(* CODESYS project boiler22.project
   Title: boiler21
   Version: 0.0.0.1

Project tree, tasks and I/O mapping:
  MyController : TM241CE40R, Schneider Electric, order no. TM241CE40R, version 4.0.2.20
    application Application
      libraries: Toolbox, 2.1.0.0 (Schneider Electric); Util, 3.5.1.0 (System); ModbusTCPIOScanner, 1.0.0.4 (Schneider Electric); SysTimeCore, 3.4.1.20 (System)
      task MAST (freewheeling, priority 1, watchdog 100 ms x 1) calls parmStore, service, main, SafeTmr
      task Analog (cyclic, interval t#100ms, priority 2) calls Analog, control
      task calcStat (cyclic, interval t#5s, priority 3) calls calcEnergy
      function HiddenPOU [ST]
      global variables GVL
      Prog/
        program main [ST]
        program Analog [FBD]
        program control [FBD]
        program SafeTmr [FBD]
        function block dualpid [ST]
        function getEnthalpy [ST]
        program service [ST]
        program calcEnergy [ST]
        function getDensity [ST]
        program parmStore [ST]
        function expo [ST]
      RecipeManager
      Symbols
      global variables PersistentVars
    DI : Digital Inputs, Schneider Electric, version 4.0.2.20
        input  xDrumLH2 : BOOL  // IDW0.I0
        input  xDrumLH1 : BOOL  // IDW0.I1
        input  xDrumLl1 : BOOL  // IDW0.I2
        input  xDrumLl2 : BOOL  // IDW0.I3
        input  xGasManOpen : BOOL  // IDW0.I4
        input  xRes1 : BOOL  // IDW0.I5
        input  xRes2 : BOOL  // IDW0.I6
        input  xDrumPh : BOOL  // IDW0.I7
        input  xGasPl : BOOL  // IDW0.I8
        input  xGasPh : BOOL  // IDW0.I9
        input  xAirPl : BOOL  // IDW0.I10
        input  xVacPl : BOOL  // IDW0.I11
        input  xBump : BOOL  // IDW0.I12
        input  xFire1 : BOOL  // IDW0.I13
        input  xTight : BOOL  // IDW0.I14
        input  xSafeOn : BOOL  // IDW0.I15
        input  xStartBn : BOOL  // IDW0.I16
        input  xStopBn : BOOL  // IDW0.I17
        input  xAlarmBn : BOOL  // IDW0.I18
        input  xGasAuto : BOOL  // IDW0.I19
        input  xTermAuto : BOOL  // IDW0.I20
        input  xPumpAuto : BOOL  // IDW0.I21
        input  xExhAuto : BOOL  // IDW0.I22
        input  xFanAuto : BOOL  // IDW0.I23
        unmapped channels: IDW0, IB1
    DQ : Digital Outputs, Schneider Electric, version 4.0.2.20
        output yTermOpen : BOOL  // QW0.Q0
        output yTermClose : BOOL  // QW0.Q1
        output ySuppOpen : BOOL  // QW0.Q2
        output ySuppClose : BOOL  // QW0.Q3
        output yCutofVal : BOOL  // QW0.Q4
        output yBurnerVal : BOOL  // QW0.Q5
        output ySafeVal : BOOL  // QW0.Q6
        output yLitherVal : BOOL  // QW0.Q7
        output yStartFan : BOOL  // QW0.Q8
        output yStartPump : BOOL  // QW0.Q9
        output yGasOpen : BOOL  // QW0.Q10
        output yGasClose : BOOL  // QW0.Q11
        output yPlcStop : BOOL  // QW0.Q12
        output yLamp : BOOL  // QW0.Q13
        output ySerena : BOOL  // QW0.Q14
        output yIgniter : BOOL  // QW0.Q15
        unmapped channels: QW0, QB1
    Counters : Counters, Schneider Electric, version 4.0.2.20
    Pulse_Generators : Pulse Generators, Schneider Electric, version 4.0.2.20
    Cartridge_1 : Cartridge, Schneider Electric, version 4.0.2.20
    Cartridge_2 : Cartridge, Schneider Electric, version 4.0.2.20
    IO_Bus : IO bus - TM3, Schneider Electric, version 4.0.2.20
      Module_2 : TM3AQ4/G, Schneider Electric, order no. TM3AQ4/G, version 1.0.0.10
          settings: KPI Configuration.KPI Configuration[0] = 19; KPI Configuration.KPI Configuration[1] = 19; KPI Configuration.KPI Configuration[2] = 19; KPI Configuration.KPI Configuration[3] = 19; KPI Configuration.KPI Configuration[5] = 0; KPI Configuration.KPI Configuration[7] = 0; KPI Configuration.KPI Configuration[9] = 0; KPI Configuration.KPI Configuration[11] = 0; KPI Configuration.KPI Configuration[12] = 160; KPI Configuration.KPI Configuration[13] = 15; KPI Configuration.KPI Configuration[14] = 160; KPI Configuration.KPI Configuration[15] = 15; KPI Configuration.KPI Configuration[16] = 160; KPI Configuration.KPI Configuration[17] = 15; KPI Configuration.KPI Configuration[18] = 160; KPI Configuration.KPI Configuration[19] = 15
          output Out1 : INT  // QW0
          output Out2 : INT  // QW1
          output Out3 : INT  // QW2
          output Out4 : INT  // QW3
          input  ibModule_2_IBStatusQW0 : BYTE  // IBStatusQW0
          input  ibModule_2_IBStatusQW1 : BYTE  // IBStatusQW1
          input  ibModule_2_IBStatusQW2 : BYTE  // IBStatusQW2
          input  ibModule_2_IBStatusQW3 : BYTE  // IBStatusQW3
      Module_3 : TM3AI8/G, Schneider Electric, order no. TM3AI8/G, version 1.0.0.12
          settings: KPI Configuration.KPI Configuration[0] = 35; KPI Configuration.KPI Configuration[1] = 35; KPI Configuration.KPI Configuration[2] = 35; KPI Configuration.KPI Configuration[3] = 35; KPI Configuration.KPI Configuration[4] = 35; KPI Configuration.KPI Configuration[5] = 35; KPI Configuration.KPI Configuration[6] = 35; KPI Configuration.KPI Configuration[7] = 35; KPI Configuration.KPI Configuration[9] = 0; KPI Configuration.KPI Configuration[11] = 0; KPI Configuration.KPI Configuration[13] = 0; KPI Configuration.KPI Configuration[15] = 0; KPI Configuration.KPI Configuration[17] = 0; KPI Configuration.KPI Configuration[19] = 0; KPI Configuration.KPI Configuration[21] = 0; KPI Configuration.KPI Configuration[23] = 0; KPI Configuration.KPI Configuration[24] = 160; KPI Configuration.KPI Configuration[25] = 15; KPI Configuration.KPI Configuration[26] = 160; KPI Configuration.KPI Configuration[27] = 15; KPI Configuration.KPI Configuration[28] = 160; KPI Configuration.KPI Configuration[29] = 15; KPI Configuration.KPI Configuration[30] = 160; KPI Configuration.KPI Configuration[31] = 15; KPI Configuration.KPI Configuration[32] = 160; KPI Configuration.KPI Configuration[33] = 15; KPI Configuration.KPI Configuration[34] = 160; KPI Configuration.KPI Configuration[35] = 15; KPI Configuration.KPI Configuration[36] = 160; KPI Configuration.KPI Configuration[37] = 15; KPI Configuration.KPI Configuration[38] = 160; KPI Configuration.KPI Configuration[39] = 15
          input  AI000 : INT  // IW0
          input  AI001 : INT  // IW1
          input  AI002 : INT  // IW2
          input  AI003 : INT  // IW3
          input  AI004 : INT  // IW4
          input  AI005 : INT  // IW5
          input  AI006 : INT  // IW6
          input  AI007 : INT  // IW7
          input  ibModule_3_IBStatusIW0 : BYTE  // IBStatusIW0
          input  ibModule_3_IBStatusIW1 : BYTE  // IBStatusIW1
          input  ibModule_3_IBStatusIW2 : BYTE  // IBStatusIW2
          input  ibModule_3_IBStatusIW3 : BYTE  // IBStatusIW3
          input  ibModule_3_IBStatusIW4 : BYTE  // IBStatusIW4
          input  ibModule_3_IBStatusIW5 : BYTE  // IBStatusIW5
          input  ibModule_3_IBStatusIW6 : BYTE  // IBStatusIW6
          input  ibModule_3_IBStatusIW7 : BYTE  // IBStatusIW7
      Module_4 : TM3AI8/G, Schneider Electric, order no. TM3AI8/G, version 1.0.0.12
          settings: KPI Configuration.KPI Configuration[0] = 35; KPI Configuration.KPI Configuration[1] = 35; KPI Configuration.KPI Configuration[2] = 35; KPI Configuration.KPI Configuration[3] = 35; KPI Configuration.KPI Configuration[4] = 35; KPI Configuration.KPI Configuration[5] = 35; KPI Configuration.KPI Configuration[6] = 35; KPI Configuration.KPI Configuration[7] = 35; KPI Configuration.KPI Configuration[9] = 0; KPI Configuration.KPI Configuration[11] = 0; KPI Configuration.KPI Configuration[13] = 0; KPI Configuration.KPI Configuration[15] = 0; KPI Configuration.KPI Configuration[17] = 0; KPI Configuration.KPI Configuration[19] = 0; KPI Configuration.KPI Configuration[21] = 0; KPI Configuration.KPI Configuration[23] = 0; KPI Configuration.KPI Configuration[24] = 160; KPI Configuration.KPI Configuration[25] = 15; KPI Configuration.KPI Configuration[26] = 160; KPI Configuration.KPI Configuration[27] = 15; KPI Configuration.KPI Configuration[28] = 160; KPI Configuration.KPI Configuration[29] = 15; KPI Configuration.KPI Configuration[30] = 160; KPI Configuration.KPI Configuration[31] = 15; KPI Configuration.KPI Configuration[32] = 160; KPI Configuration.KPI Configuration[33] = 15; KPI Configuration.KPI Configuration[34] = 160; KPI Configuration.KPI Configuration[35] = 15; KPI Configuration.KPI Configuration[36] = 160; KPI Configuration.KPI Configuration[37] = 15; KPI Configuration.KPI Configuration[38] = 160; KPI Configuration.KPI Configuration[39] = 15
          input  AI010 : INT  // IW0
          input  AI011 : INT  // IW1
          input  AI012 : INT  // IW2
          input  AI013 : INT  // IW3
          input  AI014 : INT  // IW4
          input  AI015 : INT  // IW5
          input  AI016 : INT  // IW6
          input  AI017 : INT  // IW7
          input  ibModule_4_IBStatusIW0 : BYTE  // IBStatusIW0
          input  ibModule_4_IBStatusIW1 : BYTE  // IBStatusIW1
          input  ibModule_4_IBStatusIW2 : BYTE  // IBStatusIW2
          input  ibModule_4_IBStatusIW3 : BYTE  // IBStatusIW3
          input  ibModule_4_IBStatusIW4 : BYTE  // IBStatusIW4
          input  ibModule_4_IBStatusIW5 : BYTE  // IBStatusIW5
          input  ibModule_4_IBStatusIW6 : BYTE  // IBStatusIW6
          input  ibModule_4_IBStatusIW7 : BYTE  // IBStatusIW7
      Module_5 : TM3AI8/G, Schneider Electric, order no. TM3AI8/G, version 1.0.0.12
          settings: KPI Configuration.KPI Configuration[0] = 35; KPI Configuration.KPI Configuration[1] = 35; KPI Configuration.KPI Configuration[2] = 35; KPI Configuration.KPI Configuration[3] = 35; KPI Configuration.KPI Configuration[4] = 35; KPI Configuration.KPI Configuration[5] = 35; KPI Configuration.KPI Configuration[6] = 35; KPI Configuration.KPI Configuration[7] = 35; KPI Configuration.KPI Configuration[9] = 0; KPI Configuration.KPI Configuration[11] = 0; KPI Configuration.KPI Configuration[13] = 0; KPI Configuration.KPI Configuration[15] = 0; KPI Configuration.KPI Configuration[17] = 0; KPI Configuration.KPI Configuration[19] = 0; KPI Configuration.KPI Configuration[21] = 0; KPI Configuration.KPI Configuration[23] = 0; KPI Configuration.KPI Configuration[24] = 160; KPI Configuration.KPI Configuration[25] = 15; KPI Configuration.KPI Configuration[26] = 160; KPI Configuration.KPI Configuration[27] = 15; KPI Configuration.KPI Configuration[28] = 160; KPI Configuration.KPI Configuration[29] = 15; KPI Configuration.KPI Configuration[30] = 160; KPI Configuration.KPI Configuration[31] = 15; KPI Configuration.KPI Configuration[32] = 160; KPI Configuration.KPI Configuration[33] = 15; KPI Configuration.KPI Configuration[34] = 160; KPI Configuration.KPI Configuration[35] = 15; KPI Configuration.KPI Configuration[36] = 160; KPI Configuration.KPI Configuration[37] = 15; KPI Configuration.KPI Configuration[38] = 160; KPI Configuration.KPI Configuration[39] = 15
          input  AI020 : INT  // IW0
          input  AI021 : INT  // IW1
          input  AI022 : INT  // IW2
          input  AI023 : INT  // IW3
          input  AI024 : INT  // IW4
          input  AI025 : INT  // IW5
          input  AI026 : INT  // IW6
          input  AI027 : INT  // IW7
          input  ibModule_5_IBStatusIW0 : BYTE  // IBStatusIW0
          input  ibModule_5_IBStatusIW1 : BYTE  // IBStatusIW1
          input  ibModule_5_IBStatusIW2 : BYTE  // IBStatusIW2
          input  ibModule_5_IBStatusIW3 : BYTE  // IBStatusIW3
          input  ibModule_5_IBStatusIW4 : BYTE  // IBStatusIW4
          input  ibModule_5_IBStatusIW5 : BYTE  // IBStatusIW5
          input  ibModule_5_IBStatusIW6 : BYTE  // IBStatusIW6
          input  ibModule_5_IBStatusIW7 : BYTE  // IBStatusIW7
    COM_Bus : COM bus, Schneider Electric, version 4.0.2.20
    Ethernet_1 : Ethernet Network, Schneider Electric, version 4.0.2.20
        settings: IPAddress = [192, 168, 15, 152]; SubnetMask = [255, 255, 255, 0]; GatewayAddress = [192, 168, 15, 1]; DeviceName = 'boiler2'; WebServer = FALSE; FTP Server = FALSE; SoMachine Protocol = TRUE; Modbus Server = TRUE; NetManage Protocol = FALSE; SNMP protocol = FALSE; Enable Routing = FALSE; WebVisu protocol = FALSE
    Serial_Line_1 : Serial line, Schneider Electric, version 4.0.2.20
      Modbus_Manager : Modbus Manager, Schneider Electric, version 4.0.0.2
    Serial_Line_2 : Serial line, Schneider Electric, version 4.0.2.20
      Modbus_IOScanner : Modbus IOScanner, Schneider Electric, version 3.5.3.6
        drvFan : Generic Modbus Slave, Schneider Electric, version 3.5.3.6
            settings: SlaveAddress = 12; ResponseTimeout = 1000; Channel 1.Function Code = 3; Channel 1.Read Offset = 16#0008; Channel 1.Read Length = 1; Channel 1.Write Offset = 0; Channel 1.Write Length = 0; Channel 1.Cycle Time = 0; Channel 2.Function Code = 3; Channel 2.Read Offset = 16#00C8; Channel 2.Read Length = 8; Channel 2.Write Offset = 0; Channel 2.Write Length = 0; Channel 2.Cycle Time = 0
            input  fanStatus : WORD  // Channel 1.Channel 1[0]
            input  fan0 : WORD  // Channel 2.Channel 2[0]
            input  fan1 : WORD  // Channel 2.Channel 2[1]
            input  fan2 : WORD  // Channel 2.Channel 2[2]
            input  fan3 : WORD  // Channel 2.Channel 2[3]
            input  fan4 : WORD  // Channel 2.Channel 2[4]
            input  fan5 : WORD  // Channel 2.Channel 2[5]
            input  fan6 : WORD  // Channel 2.Channel 2[6]
            input  fan7 : WORD  // Channel 2.Channel 2[7]
            unmapped channels: Channel 1, Channel 2
        PD150 : Generic Modbus Slave, Schneider Electric, version 3.5.3.6
            settings: SlaveAddress = 16; ResponseTimeout = 1000; Channel 1.Function Code = 3; Channel 1.Read Offset = 16#0013; Channel 1.Read Length = 2; Channel 1.Write Offset = 0; Channel 1.Write Length = 0; Channel 1.Cycle Time = 0
            input  pdi1 : WORD  // Channel 1.Channel 1[0]
            input  pdi2 : WORD  // Channel 1.Channel 1[1]
            unmapped channels: Channel 1
        drvPump : Generic Modbus Slave, Schneider Electric, version 3.5.3.6
            settings: SlaveAddress = 10; ResponseTimeout = 1000; Channel 1.Function Code = 3; Channel 1.Read Offset = 16#0066; Channel 1.Read Length = 8; Channel 1.Write Offset = 0; Channel 1.Write Length = 0; Channel 1.Cycle Time = 0; Channel 2.Function Code = 2; Channel 2.Read Offset = 16#0000; Channel 2.Read Length = 16; Channel 2.Write Offset = 0; Channel 2.Write Length = 0; Channel 2.Cycle Time = 0
            input  pump0 : WORD  // Channel 1.Channel 1[0]
            input  pump1 : WORD  // Channel 1.Channel 1[1]
            input  pump2 : WORD  // Channel 1.Channel 1[2]
            input  pump3 : WORD  // Channel 1.Channel 1[3]
            input  pump4 : WORD  // Channel 1.Channel 1[4]
            input  pump5 : WORD  // Channel 1.Channel 1[5]
            input  pump6 : WORD  // Channel 1.Channel 1[6]
            input  pump7 : WORD  // Channel 1.Channel 1[7]
            input  pumpRun : BOOL  // Channel 2.Channel 2[0].Bit2
            unmapped channels: Channel 1, Channel 2
        drvExh : Generic Modbus Slave, Schneider Electric, version 3.5.3.6
            settings: SlaveAddress = 11; ResponseTimeout = 1000; Channel 1.Function Code = 3; Channel 1.Read Offset = 16#1101; Channel 1.Read Length = 11; Channel 1.Write Offset = 0; Channel 1.Write Length = 0; Channel 1.Cycle Time = 0; Channel 2.Function Code = 3; Channel 2.Read Offset = 16#2100; Channel 2.Read Length = 3; Channel 2.Write Offset = 0; Channel 2.Write Length = 0; Channel 2.Cycle Time = 0
            input  exh0 : WORD  // Channel 1.Channel 1[0]
            input  exh1 : WORD  // Channel 1.Channel 1[1]
            input  exh2 : WORD  // Channel 1.Channel 1[2]
            input  exh3 : WORD  // Channel 1.Channel 1[3]
            input  exh4 : WORD  // Channel 1.Channel 1[4]
            input  exh5 : WORD  // Channel 1.Channel 1[5]
            input  exh6 : WORD  // Channel 1.Channel 1[6]
            input  exh7 : WORD  // Channel 1.Channel 1[7]
            input  exh8 : WORD  // Channel 1.Channel 1[8]
            input  exh9 : WORD  // Channel 1.Channel 1[9]
            input  exh10 : WORD  // Channel 1.Channel 1[10]
            input  exhStatus : WORD  // Channel 2.Channel 2[0]
            unmapped channels: Channel 1, Channel 2
  FdtConnections : FDT Connections, Schneider Electric, version 1.0.0.2
    Modbus_Serial_Line_Manager : Modbus Serial Line Manager, Schneider Electric, version 2.2.5
*)

// MyController/Application/GVL

VAR_GLOBAL
allAM AT %MW0: INT;

AM001 AT %MX0.0: BOOL;
AM002 AT %MX0.1: BOOL;
AM003 AT %MX0.2: BOOL;
AM004 AT %MX0.3: BOOL;
AM005 AT %MX0.4: BOOL;
AM006 AT %MX0.5: BOOL;
AM007 AT %MX0.6: BOOL;
AM008 AT %MX0.7: BOOL;

amGas AT %MX2.0: BOOL := true;
amTerm AT %MX2.1: BOOL := true;
amSupp AT %MX2.2: BOOL := true;

Alm0001 AT %MX4.0: BOOL;
Alm0002 AT %MX4.1: BOOL;
Alm0003 AT %MX4.2: BOOL;
Alm0004 AT %MX4.3: BOOL;
Alm0005 AT %MX4.4: BOOL;
Alm0006 AT %MX4.5: BOOL;
Alm0007 AT %MX4.6: BOOL;
Alm0008 AT %MX4.7: BOOL;
Alm0009 AT %MX5.0: BOOL;
Alm0010 AT %MX5.1: BOOL;
Alm0011 AT %MX5.2: BOOL;
Alm0012 AT %MX5.3: BOOL;
alFire1 AT %MX5.4: BOOL;
alFan AT %MX5.5: BOOL;
alExh AT %MX5.6: BOOL;
alPump AT %MX5.7: BOOL;


alSupport AT %MX6.0: BOOL;
linkPump AT %MX6.1: BOOL;
linkFan AT %MX6.2: BOOL;
linkExh AT %MX6.3: BOOL;
linkPD150 AT %MX6.4: BOOL;
stab1 AT %MX6.5: BOOL;
stab2 AT %MX6.6: BOOL;
stab3 AT %MX6.7: BOOL;
stab4 AT %MX7.0: BOOL;
stab5 AT %MX7.1: BOOL;
xFanRun AT %MX7.2: BOOL;
xExhRun AT %MX7.3: BOOL;
xPumpRun AT %MX7.4: BOOL;
stWait AT %MX7.5: BOOL;
Alert AT %MX7.6: BOOL;
Halt AT %MX7.7: BOOL;

// це треба буде писати зверху
Run AT %MX8.0: BOOL;
Cvit AT %MX10.0: BOOL;
prLock AT %MX12.0: BOOL;
serenaLock AT %MX12.1: BOOL;

bnAll AT %MW7: INT;
bnStart AT %MX14.0: BOOL;
bnStop AT %MX14.1: BOOL;
// список прогодження кроків програми запуску
check0 AT %MX16.0: BOOL;
check1 AT %MX16.1: BOOL;
check2 AT %MX16.2: BOOL;
check3 AT %MX16.3: BOOL;
check4 AT %MX16.4: BOOL;
check5 AT %MX16.5: BOOL;
check6 AT %MX16.6: BOOL;
check7 AT %MX16.7: BOOL;
check8 AT %MX17.0: BOOL;
check9 AT %MX17.1: BOOL;
check10 AT %MX17.2: BOOL;
check11 AT %MX17.3: BOOL;
check12 AT %MX17.4: BOOL;
check13 AT %MX17.5: BOOL;
check14 AT %MX17.6: BOOL;
check15 AT %MX17.7: BOOL;

checkList AT %MW8: UINT;


Pack_lo AT %MW998: WORD;
Pack_hi AT %MW999: WORD;
Pack_v AT %MD499: REAL;

Fgas AT %MD5: REAL;
Fpara AT %MD6: REAL;
Fwater AT %MD7: REAL;
Fair AT %MD8: REAL;
Ldrum AT %MD9: REAL;
Pg15a AT %MD10: REAL;
Ppara AT %MD11: REAL;
Pp7a AT %MD12: REAL;
Tpar AT %MD13: REAL;
Tv3a AT %MD14: REAL;
Tv4a AT %MD15: REAL;
Tk AT %MD16: REAL;
Ta5a AT %MD17: REAL;
Ta6a AT %MD18: REAL;
Tp17a AT %MD19: REAL;
Tp18a AT %MD20: REAL;
Pair AT %MD21: REAL;
Pvac AT %MD22: REAL;
Pv12a AT %MD23: REAL;
gGas AT %MD24: REAL;
gTerm AT %MD25: REAL;
gSupp AT %MD26: REAL;
QO2fume AT %MD27: REAL;
Vx AT %MD28: REAL;

W01 AT %MW10: WORD;
W02 AT %MW11: WORD;

END_VAR

VAR_GLOBAL RETAIN
cPump AT %MD29: REAL;
cFan AT %MD30: REAL;
cExh AT %MD31: REAL;
cGas AT %MD32: REAL;
cTerm AT %MD33: REAL;
cSupport AT %MD34: REAL;
cX AT %MD35: REAL;
END_VAR

VAR_GLOBAL
FanSpeed AT %MD36: REAL;
FanCurrent AT %MD37: REAL;
FanVoltage AT %MD38: REAL;
FanDC AT %MD39: REAL;
PumpSpeed AT %MD40: REAL;
PumpCurrent AT %MD41: REAL;
PumpVoltage AT %MD42: REAL;
PumpDC AT %MD43: REAL;
ExhSpeed AT %MD44: REAL;
ExhCurrent AT %MD45: REAL;
ExhVoltage AT %MD46: REAL;
ExhDC AT %MD47: REAL;

END_VAR

VAR_GLOBAL RETAIN
Sp0001 AT %MD48: REAL;
Sp0002 AT %MD49: REAL;
Sp0003 AT %MD50: REAL;
Sp0004 AT %MD51: REAL;
Sp0005 AT %MD52: REAL;
Sp0006 AT %MD53: REAL;
Sp0007 AT %MD54: REAL;
Sp0008 AT %MD55: REAL;
Sp0009 AT %MD56: REAL;
Sp0010 AT %MW114: UINT;
END_VAR

VAR_GLOBAL


// Кінцевий автомат управління котлом
State AT %MW115: UINT;
stateTight AT %MW116: UINT;
flame AT %MW117: UINT;

pvTVentPre AT %MD400: DWORD;
pvTBlowing AT %MD401: DWORD;
pvFiring AT %MD402: DWORD;
pvStartfeed AT %MD403: DWORD;
pvStartExh AT %MD404: DWORD;
pvStartfan AT %MD405: DWORD;
pvIgniting AT %MD406: DWORD;
pvTVentPost AT %MD407: DWORD;

END_VAR

VAR_GLOBAL RETAIN
backup AT %MW118: UINT;

uptime AT %MD425: REAL;
allPara AT %MD426: REAL;
allGas AT %MD427: REAL;
allWarm AT %MD428: REAL;
allEce AT %MD429: REAL;
hourPara AT %MD430: REAL;
hourGas AT %MD431: REAL;
hourWarm AT %MD432: REAL;
hourEce AT %MD433: REAL;

 
fA000 AT %MW177: UINT;
fA001 AT %MW178: UINT;
fA002 AT %MW179: UINT;
fA003 AT %MW180: UINT;
fA004 AT %MW181: UINT;
fA005 AT %MW182: UINT;
fA006 AT %MW183: UINT;
fA007 AT %MW184: UINT;
fA010 AT %MW185: UINT;
fA011 AT %MW186: UINT;
fA012 AT %MW187: UINT;
fA013 AT %MW188: UINT;
fA014 AT %MW189: UINT;
fA015 AT %MW190: UINT;
fA016 AT %MW191: UINT;
fA017 AT %MW192: UINT;
fA020 AT %MW193: UINT;
fA021 AT %MW194: UINT;
fA022 AT %MW195: UINT;
fA023 AT %MW196: UINT;
fA024 AT %MW197: UINT;
fA025 AT %MW198: UINT;
fA026 AT %MW199: UINT;
fA027 AT %MW200: UINT;

modeGas AT %MW201: UINT;

Kp0001 AT %MD101: REAL;
Ti0001 AT %MD102: REAL;
Td0001 AT %MD103: REAL;
Xmin0001 AT %MD104: REAL;
Xmax0001 AT %MD105: REAL;
Kp0002 AT %MD106: REAL;
Ti0002 AT %MD107: REAL;
Td0002 AT %MD108: REAL;
Xmin0002 AT %MD109: REAL;
Xmax0002 AT %MD110: REAL;
Kp0003 AT %MD111: REAL;
Ti0003 AT %MD112: REAL;
Td0003 AT %MD113: REAL;
Xmin0003 AT %MD114: REAL;
Xmax0003 AT %MD115: REAL;
Kp0004 AT %MD116: REAL;
Ti0004 AT %MD117: REAL;
Td0004 AT %MD118: REAL;
Xmin0004 AT %MD119: REAL;
Xmax0004 AT %MD120: REAL;
Kp0005 AT %MD121: REAL;
Ti0005 AT %MD122: REAL;
Td0005 AT %MD123: REAL;
Xmin0005 AT %MD124: REAL;
Xmax0005 AT %MD125: REAL;
Kp0006 AT %MD126: REAL;
Ti0006 AT %MD127: REAL;
Td0006 AT %MD128: REAL;
Xmin0006 AT %MD129: REAL;
Xmax0006 AT %MD130: REAL;
Kp0007 AT %MD131: REAL;
Ti0007 AT %MD132: REAL;
Td0007 AT %MD133: REAL;
Xmin0007 AT %MD134: REAL;
Xmax0007 AT %MD135: REAL;
Kp0008 AT %MD136: REAL;
Ti0008 AT %MD137: REAL;
Td0008 AT %MD138: REAL;
Xmin0008 AT %MD139: REAL;
Xmax0008 AT %MD140: REAL;
startSP0002 AT %MD141: REAL;

tMeoTerm AT %MD142: REAL;
tMeoGas AT %MD143: REAL;
dGas AT %MD144: REAL;
dTerm AT %MD145: REAL;
dSupport AT %MD146: REAL;
maxS1 AT %MD147: REAL;
maxS2 AT %MD148: REAL;
maxS3 AT %MD149: REAL;
maxS4 AT %MD150: REAL;
maxS5 AT %MD151: REAL;
K2001 AT %MD152: REAL;
startPump AT %MD153: REAL;
startFan AT %MD154: REAL;
startExh AT %MD155: REAL;
startGas AT %MD156: REAL;
startTerm AT %MD157: REAL;
gOffset AT %MD158: REAL;
gGain AT %MD159: REAL;
heatingGas AT %MD160: REAL;
sca_Ppara AT %MD161: REAL;
max_Ppara AT %MD162: REAL;
sca_Tpar AT %MD163: REAL;
max_Tpar AT %MD164: REAL;
sca_Tv3a AT %MD165: REAL;
max_Tv3a AT %MD166: REAL;
sca_Fgas AT %MD167: REAL;
max_Fgas AT %MD168: REAL;
sca_Fpara AT %MD169: REAL;
max_Fpara AT %MD170: REAL;
qgas AT %MD171: REAL;
sca_Fwater AT %MD172: REAL;
max_Fwater AT %MD173: REAL;
gTermOffset AT %MD174: REAL;
gTermGain AT %MD175: REAL;
gSuppOffset AT %MD176: REAL;
gSuppGain AT %MD177: REAL;
Ke0001 AT %MD178: REAL;
Ke0002 AT %MD179: REAL;
Ke0003 AT %MD180: REAL;
Ke0004 AT %MD181: REAL;
Ke0005 AT %MD182: REAL;
Kmix001 AT %MD183: REAL;
Kmix002 AT %MD184: REAL;
Kmix003 AT %MD185: REAL;
Kmix004 AT %MD186: REAL;
Kmix005 AT %MD187: REAL;
Omix001 AT %MD188: REAL;
Omix002 AT %MD189: REAL;
Omix003 AT %MD190: REAL;
Omix004 AT %MD191: REAL;
Omix005 AT %MD192: REAL;
ignSP0002 AT %MD193: REAL;

Tpr0001 AT %MD256: DWORD;
Tpr0002 AT %MD257: DWORD;
Tpr0003 AT %MD258: DWORD;
Tpr0004 AT %MD259: DWORD;
Tpr0005 AT %MD260: DWORD;
Tpr0006 AT %MD261: DWORD;
Tpr0007 AT %MD262: DWORD;
Tpr0008 AT %MD263: DWORD;
Tpr0009 AT %MD264: DWORD;
Tpr0010 AT %MD265: DWORD;
Tpr0011 AT %MD266: DWORD;
Tpr0012 AT %MD267: DWORD;
spTstart AT %MD268: DWORD;
spTVentPre AT %MD269: DWORD;
spTVentPost AT %MD270: DWORD;
spTBlowing AT %MD271: DWORD;
spStartfeed AT %MD272: DWORD;
spStartExh AT %MD273: DWORD;
spStartfan AT %MD274: DWORD;
spIgniting AT %MD275: DWORD;



END_VAR

VAR_GLOBAL
firstStep: BOOL:=TRUE;
	
Xt0001: REAL;
Xt0002: REAL;
Xt0003: REAL;
Xt0004: REAL;
Xt0005: REAL;
Xt0006: REAL;
Xt0007: REAL;
Xt0008: REAL;

tMeo1: TIME;
tMeo2: TIME;
tMeo3: TIME;

enthalpy: REAL;

regO2en: BOOL;
pwmParam: stPwmPara;

p4GasOpen: BOOL;
p4GasClose: BOOL;

END_VAR

VAR_GLOBAL CONSTANT
// таблиця ентальпії пари від 200 до 500 *С з кроком 10*С і від 1000 до 3000 кПа з кроком 500кПа	
enthalpyTab: ARRAY[0..30] OF ARRAY[0..4] OF REAL := [
[2827.5,2795.3,852.6,852.8,853.0],
[2851.5,2822.9,897.8,898.1,898.1],
[2874.9,2849.2,2820.4,943.7,943.9],
[2897.9,2874.7,2849.0,2820.4,990.3],
[2920.5,2899.3,2876.3,2851.0,2823.0],
[2942.8,2923.4,2902.5,2879.9,2855.2],
[2964.8,2947.0,2927.9,2907.5,2885.5],
[2986.7,2970.2,2952.7,2934.1,2914.2],
[3008.3,2993.0,2976.9,2959.8,2941.8],
[3029.9,3015.6,3000.6,2984.9,2968.4],
[3051.3,3037.9,3024.0,3009.4,2994.2],
[3072.7,3060.1,3047.0,3033.4,3019.3],
[3094.0,3082.1,3069.8,3057.1,3044.0],
[3115.3,3104.0,3092.4,3080.5,3068.2],
[3136.5,3125.8,3114.9,3103.6,3092.1],
[3157.7,3147.6,3137.2,3126.6,3115.7],
[3178.9,3169.3,3159.5,3149.6,3139.3],
[3200.2,3191.1,3181.8,3172.4,3162.7],
[3221.5,3212.8,3204.0,3195.0,3185.8],
[3242.8,3234.5,3226.1,3217.5,3208.8],
[3264.0,3256.1,3248.1,3239.9,3231.6],
[3285.3,3277.7,3270.0,3262.2,3254.3],
[3306.6,3299.3,3291.9,3284.5,3276.9],
[3327.9,3320.9,3313.8,3306.7,3299.4],
[3349.3,3342.6,3335.7,3328.9,3321.9],
[3370.7,3364.2,3357.7,3351.0,3344.4],
[3392.1,3385.9,3379.6,3373.2,3366.8],
[3413.8,3407.6,3401.5,3395.4,3389.2],
[3435.1,3429.3,3423.5,3417.5,3411.6],
[3456.7,3451.1,3445.4,3439.7,3434.0],
[3478.3,3472.9,3467.4,3461.9,3456.4]
];	
// питомий обёєм 
spvolTab: ARRAY[0..30] OF ARRAY[0..4] OF REAL := [
[	0.2059	,	0.1324	,	0.001156	,	0.0011555	,	0.001155	],
[	0.2115	,	0.1366	,	0.0011725	,	0.0011719	,	0.0011714	],
[	0.2169	,	0.14	,	0.10211	,	0.0011897	,	0.0011891	],
[	0.2223	,	0.1445	,	0.1053	,	0.08164	,	0.0012084	],
[	0.2275	,	0.1483	,	0.1084	,	0.08439	,	0.06818	],
[	0.2327	,	0.152	,	0.1115	,	0.08701	,	0.07058	],
[	0.2378	,	0.1556	,	0.1144	,	0.08953	,	0.07286	],
[	0.2429	,	0.1592	,	0.1172	,	0.09197	,	0.07504	],
[	0.248	,	0.1627	,	0.12	,	0.09434	,	0.07714	],
[	0.253	,	0.1662	,	0.1228	,	0.09665	,	0.07918	],
[	0.258	,	0.1697	,	0.1255	,	0.09892	,	0.08116	],
[	0.2629	,	0.1731	,	0.1282	,	0.10114	,	0.0831	],
[	0.2678	,	0.1765	,	0.1308	,	0.10334	,	0.085	],
[	0.2727	,	0.1799	,	0.1334	,	0.1055	,	0.08687	],
[	0.2776	,	0.1832	,	0.136	,	0.1076	,	0.08871	],
[	0.2825	,	0.1866	,	0.1386	,	0.1098	,	0.09053	],
[	0.2873	,	0.1899	,	0.1411	,	0.1119	,	0.09232	],
[	0.2921	,	0.1932	,	0.1436	,	0.1139	,	0.0941	],
[	0.297	,	0.1964	,	0.1462	,	0.116	,	0.09586	],
[	0.3018	,	0.1997	,	0.1487	,	0.118	,	0.0976	],
[	0.3066	,	0.203	,	0.1512	,	0.1201	,	0.09933	],
[	0.3113	,	0.2062	,	0.1536	,	0.1221	,	0.10105	],
[	0.3161	,	0.2095	,	0.1561	,	0.1241	,	0.10276	],
[	0.3209	,	0.2127	,	0.1586	,	0.1261	,	0.1045	],
[	0.3256	,	0.2159	,	0.161	,	0.1281	,	0.1061	],
[	0.3304	,	0.2191	,	0.1635	,	0.1301	,	0.1078	],
[	0.3351	,	0.2223	,	0.1659	,	0.1321	,	0.1095	],
[	0.3399	,	0.2255	,	0.1684	,	0.134	,	0.1112	],
[	0.3446	,	0.2287	,	0.1708	,	0.136	,	0.1128	],
[	0.3493	,	0.2319	,	0.1732	,	0.138	,	0.1145	],
[	0.354	,	0.2351	,	0.1756	,	0.1399	,	0.1161	]
];
densityTab: ARRAY[0..30] OF ARRAY[0..4] OF REAL := [	
[ 4.85672656629432 , 7.55287009063444 , 865.051903114187 , 865.426222414539 , 865.800865800866 ],
[ 4.72813238770686 , 7.32064421669107 , 852.878464818763 , 853.315129277242 , 853.679358033123 ],
[ 4.61041954817888 , 7.14285714285714 , 9.79336010185095 , 840.548037320333 , 840.972163821377 ],
[ 4.49842555105713 , 6.92041522491349 , 9.49667616334283 , 12.2488975992161 , 827.540549486925 ],
[ 4.3956043956044 , 6.74308833445718 , 9.22509225092251 , 11.8497452304775 , 14.6670577882077 ],
[ 4.29737859905458 , 6.57894736842105 , 8.96860986547085 , 11.4929318469141 , 14.168319637291 ],
[ 4.20521446593776 , 6.426735218509 , 8.74125874125874 , 11.1694404110354 , 13.7249519626681 ],
[ 4.11692054343351 , 6.28140703517588 , 8.53242320819113 , 10.873110796999 , 13.3262260127932 ],
[ 4.03225806451613 , 6.14628149969269 , 8.33333333333333 , 10.5999576001696 , 12.9634430904848 ],
[ 3.95256916996047 , 6.01684717208183 , 8.14332247557003 , 10.3466114847387 , 12.6294518817883 ],
[ 3.87596899224806 , 5.89275191514437 , 7.96812749003984 , 10.1091791346543 , 12.3213405618531 ],
[ 3.80372765310004 , 5.77700751010976 , 7.8003120124805 , 9.8872849515523 , 12.0336943441637 ],
[ 3.73412994772218 , 5.6657223796034 , 7.64525993883792 , 9.67679504548094 , 11.7647058823529 ],
[ 3.66703337000367 , 5.55864369093941 , 7.49625187406297 , 9.47867298578199 , 11.5114538966271 ],
[ 3.60230547550432 , 5.4585152838428 , 7.35294117647059 , 9.29368029739777 , 11.2726862811408 ],
[ 3.53982300884956 , 5.35905680600214 , 7.21500721500721 , 9.10746812386157 , 11.0460620788689 ],
[ 3.48068221371389 , 5.26592943654555 , 7.0871722182849 , 8.93655049151028 , 10.8318890814558 ],
[ 3.42348510783978 , 5.175983436853 , 6.96378830083565 , 8.77963125548727 , 10.6269925611052 ],
[ 3.36700336700337 , 5.09164969450102 , 6.83994528043776 , 8.62068965517241 , 10.4318798247444 ],
[ 3.31345261762757 , 5.00751126690035 , 6.72494956287828 , 8.47457627118644 , 10.2459016393443 ],
[ 3.26157860404436 , 4.92610837438424 , 6.61375661375661 , 8.32639467110741 , 10.067451927917 ],
[ 3.2123353678124 , 4.84966052376334 , 6.51041666666667 , 8.19000819000819 , 9.8960910440376 ],
[ 3.16355583676052 , 4.77326968973747 , 6.40614990390775 , 8.058017727639 , 9.73141300116777 ],
[ 3.11623558741041 , 4.70145745181006 , 6.30517023959647 , 7.93021411578112 , 9.56937799043062 ],
[ 3.07125307125307 , 4.63177396943029 , 6.2111801242236 , 7.8064012490242 , 9.42507068803016 ],
[ 3.02663438256659 , 4.56412596987677 , 6.11620795107034 , 7.68639508070715 , 9.27643784786642 ],
[ 2.98418382572366 , 4.49842555105713 , 6.02772754671489 , 7.57002271006813 , 9.1324200913242 ],
[ 2.94204177699323 , 4.43458980044346 , 5.93824228028504 , 7.46268656716418 , 8.99280575539568 ],
[ 2.90191526407429 , 4.37254044599913 , 5.85480093676815 , 7.35294117647059 , 8.86524822695035 ],
[ 2.86286859433152 , 4.3122035360069 , 5.77367205542725 , 7.2463768115942 , 8.73362445414847 ],
[ 2.82485875706215 , 4.25350914504466 , 5.69476082004556 , 7.14796283059328 , 8.61326442721792 ]
];
// вектор температури
termTab: ARRAY[0..30] OF REAL := [
200.0	,
210.0	,
220.0	,
230.0	,
240.0	,
250.0	,
260.0	,
270.0	,
280.0	,
290.0	,
300.0 ,
310.0	,
320.0	,
330.0	,
340.0	,
350.0	,
360.0	,
370.0	,
380.0	,
390.0	,
400.0	,
410.0	,
420.0	,
430.0	,
440.0	,
450.0	,
460.0	,
470.0	,
480.0	,
490.0	,
500.0	];

// вектор тиску
preshTab: ARRAY[0..4] OF REAL :=[1000.0,1500.0,2000.0,2500.0,3000.0];
// векторентальпії води 90 100 110 *С
enthalpyWater: ARRAY[0..2] OF REAL :=[378.4,420.5,462.7];
// константа перерахунку для прив,ящки до часу = 1/3600000/2 
timeSlot: REAL:=1.3888888889E-7 ; 

ST_STOP: UINT:=0;
ST_WAIT: UINT:=1;
ST_TESTSERENA: UINT:=2;
ST_STARTFEED: UINT:=3;
ST_STARTEXH: UINT:=4;
ST_CHECKTIGHT: UINT:=5;
ST_STARTFAN: UINT:=6;
ST_VENTILATION: UINT:=7;
ST_BLOWING: UINT:=8;
ST_PREPARE: UINT:=9;
ST_IGNITING: UINT:=10;
ST_FIRING: UINT:=11;
ST_HEATING: UINT:=12;
ST_RUN: UINT:=13;
ST_SHUTDOWN: UINT:=14;
ST_FAIL: UINT:=15;

spFiring: TIME:=T#15S;

END_VAR

// MyController/Application/PersistentVars
VAR_GLOBAL PERSISTENT RETAIN

bakfA000: UINT;
bakfA001: UINT;
bakfA002: UINT;
bakfA003: UINT;
bakfA004: UINT;
bakfA005: UINT;
bakfA006: UINT;
bakfA007: UINT;
bakfA010: UINT;
bakfA011: UINT;
bakfA012: UINT;
bakfA013: UINT;
bakfA014: UINT;
bakfA015: UINT;
bakfA016: UINT;
bakfA017: UINT;
bakfA020: UINT;
bakfA021: UINT;
bakfA022: UINT;
bakfA023: UINT;
bakfA024: UINT;
bakfA025: UINT;
bakfA026: UINT;
bakfA027: UINT;
bakmodeGas: UINT;

bakSp0001: REAL;
bakKp0001: REAL;
bakTi0001: REAL;
bakTd0001: REAL;
bakXmin0001: REAL;
bakXmax0001: REAL;
bakSp0002: REAL;
bakKp0002: REAL;
bakTi0002: REAL;
bakTd0002: REAL;
bakXmin0002: REAL;
bakXmax0002: REAL;
bakSp0003: REAL;
bakKp0003: REAL;
bakTi0003: REAL;
bakTd0003: REAL;
bakXmin0003: REAL;
bakXmax0003: REAL;
bakSp0004: REAL;
bakKp0004: REAL;
bakTi0004: REAL;
bakTd0004: REAL;
bakXmin0004: REAL;
bakXmax0004: REAL;
bakSp0005: REAL;
bakKp0005: REAL;
bakTi0005: REAL;
bakTd0005: REAL;
bakXmin0005: REAL;
bakXmax0005: REAL;
bakSp0006: REAL;
bakKp0006: REAL;
bakTi0006: REAL;
bakTd0006: REAL;
bakXmin0006: REAL;
bakXmax0006: REAL;
bakSp0007: REAL;
bakKp0007: REAL;
bakTi0007: REAL;
bakTd0007: REAL;
bakXmin0007: REAL;
bakXmax0007: REAL;
baktMeoTerm: REAL;
baktMeoGas: REAL;
bakdGas: REAL;
bakdTerm: REAL;
bakdSupp: REAL;
bakmaxS1: REAL;
bakmaxS2: REAL;
bakmaxS3: REAL;
bakmaxS4: REAL;
bakmaxS5: REAL;
bakK2001: REAL;
bakstartPump: REAL;
bakstartFan: REAL;
bakstartExh: REAL;
bakstartGas: REAL;
bakstartTerm: REAL;
bakgOffset: REAL;
bakgGain: REAL;
bakheatingGas: REAL;
baksca_Ppara: REAL;
bakmax_Ppara: REAL;
baksca_Tpar: REAL;
bakmax_Tpar: REAL;
baksca_Tv3a: REAL;
bakmax_Tv3a: REAL;
baksca_Fgas: REAL;
bakmax_Fgas: REAL;
baksca_Fpara: REAL;
bakmax_Fpara: REAL;
bakqgas: REAL;
baksca_Fwater: REAL;
bakmax_Fwater: REAL;
bakgTermOffset: REAL;
bakgTermGain: REAL;
bakgSuppOffset: REAL;
bakgSuppGain: REAL;

bakTpr0001: DWORD;
bakTpr0002: DWORD;
bakTpr0003: DWORD;
bakTpr0004: DWORD;
bakTpr0005: DWORD;
bakTpr0006: DWORD;
bakTpr0007: DWORD;
bakTpr0008: DWORD;
bakTpr0009: DWORD;
bakTpr0010: DWORD;
bakTpr0011: DWORD;
bakTpr0012: DWORD;
bakspTstart: DWORD;
bakspTVentPre: DWORD;
bakspTVentPost: DWORD;
bakspTBlowing: DWORD;
bakspStartfeed: DWORD;
bakspStartExh: DWORD;
bakspStartfan: DWORD;
bakspIgniting: DWORD;

bakallPara: REAL;
bakallGas: REAL;
bakallWarm: REAL;
bakallEce: REAL;
bakhourPara: REAL;
bakhourGas: REAL;
bakhourWarm: REAL;
bakhourEce: REAL;

bakKe0001: REAL;
bakKe0002: REAL;
bakKe0003: REAL;
bakKe0004: REAL;
bakKe0005: REAL;

bakKmix001: REAL;
bakKmix002: REAL;
bakKmix003: REAL;
bakKmix004: REAL;
bakKmix005: REAL;
bakOmix001: REAL;
bakOmix002: REAL;
bakOmix003: REAL;
bakOmix004: REAL;
bakOmix005: REAL;


bakSp0008: REAL;
bakSp0009: REAL;
bakSp0010: REAL;

bakKp0008: REAL;
bakTi0008: REAL;
bakTd0008: REAL;
bakXmin0008: REAL;
bakXmax0008: REAL;
bakStartSP0002: REAL;
bakignSP0002 : REAL;

END_VAR

// MyController/Application/Prog/parmStore
PROGRAM parmStore
VAR
END_VAR

IF firstStep THEN
	IF backup=0 THEN
fA000:=bakfA000;
fA001:=bakfA001;
fA002:=bakfA002;
fA003:=bakfA003;
fA004:=bakfA004;
fA005:=bakfA005;
fA006:=bakfA006;
fA007:=bakfA007;
fA010:=bakfA010;
fA011:=bakfA011;
fA012:=bakfA012;
fA013:=bakfA013;
fA014:=bakfA014;
fA015:=bakfA015;
fA016:=bakfA016;
fA017:=bakfA017;
fA020:=bakfA020;
fA021:=bakfA021;
fA022:=bakfA022;
fA023:=bakfA023;
fA024:=bakfA024;
fA025:=bakfA025;
fA026:=bakfA026;
fA027:=bakfA027;
modeGas:=bakmodeGas;

Sp0001:=bakSp0001;
Kp0001:=bakKp0001;
Ti0001:=bakTi0001;
Td0001:=bakTd0001;
Xmin0001:=bakXmin0001;
Xmax0001:=bakXmax0001;
Sp0002:=bakSp0002;
Kp0002:=bakKp0002;
Ti0002:=bakTi0002;
Td0002:=bakTd0002;
Xmin0002:=bakXmin0002;
Xmax0002:=bakXmax0002;
Sp0003:=bakSp0003;
Kp0003:=bakKp0003;
Ti0003:=bakTi0003;
Td0003:=bakTd0003;
Xmin0003:=bakXmin0003;
Xmax0003:=bakXmax0003;
Sp0004:=bakSp0004;
Kp0004:=bakKp0004;
Ti0004:=bakTi0004;
Td0004:=bakTd0004;
Xmin0004:=bakXmin0004;
Xmax0004:=bakXmax0004;
Sp0005:=bakSp0005;
Kp0005:=bakKp0005;
Ti0005:=bakTi0005;
Td0005:=bakTd0005;
Xmin0005:=bakXmin0005;
Xmax0005:=bakXmax0005;
Sp0006:=bakSp0006;
Kp0006:=bakKp0006;
Ti0006:=bakTi0006;
Td0006:=bakTd0006;
Xmin0006:=bakXmin0006;
Xmax0006:=bakXmax0006;
Sp0007:=bakSp0007;
Kp0007:=bakKp0007;
Ti0007:=bakTi0007;
Td0007:=bakTd0007;
Xmin0007:=bakXmin0007;
Xmax0007:=bakXmax0007;
tMeoTerm:=baktMeoTerm;
tMeoGas:=baktMeoGas;
dGas:=bakdGas;
dTerm:=bakdTerm;
dSupport:=bakdSupp;
maxS1:=bakmaxS1;
maxS2:=bakmaxS2;
maxS3:=bakmaxS3;
maxS4:=bakmaxS4;
maxS5:=bakmaxS5;
K2001:=bakK2001;
startPump:=bakstartPump;
startFan:=bakstartFan;
startExh:=bakstartExh;
startGas:=bakstartGas;
startTerm:=bakstartTerm;
gOffset:=bakgOffset;
gGain:=bakgGain;
heatingGas:=bakheatingGas;
sca_Ppara:=baksca_Ppara;
max_Ppara:=bakmax_Ppara;
sca_Tpar:=baksca_Tpar;
max_Tpar:=bakmax_Tpar;
sca_Tv3a:=baksca_Tv3a;
max_Tv3a:=bakmax_Tv3a;
sca_Fgas:=baksca_Fgas;
max_Fgas:=bakmax_Fgas;
sca_Fpara:=baksca_Fpara;
max_Fpara:=bakmax_Fpara;
qgas:=bakqgas;
sca_Fwater:=baksca_Fwater;
max_Fwater:=bakmax_Fwater;
gTermOffset:=bakgTermOffset;
gTermGain:=bakgTermGain;
gSuppOffset:=bakgSuppOffset;
gSuppGain:=bakgSuppGain;

Tpr0001:=bakTpr0001;
Tpr0002:=bakTpr0002;
Tpr0003:=bakTpr0003;
Tpr0004:=bakTpr0004;
Tpr0005:=bakTpr0005;
Tpr0006:=bakTpr0006;
Tpr0007:=bakTpr0007;
Tpr0008:=bakTpr0008;
Tpr0009:=bakTpr0009;
Tpr0010:=bakTpr0010;
Tpr0011:=bakTpr0011;
Tpr0012:=bakTpr0012;
spTstart:=bakspTstart;
spTVentPre:=bakspTVentPre;
spTVentPost:=bakspTVentPost;
spTBlowing:=bakspTBlowing;
spStartfeed:=bakspStartfeed;
spStartExh:=bakspStartExh;
spStartfan:=bakspStartfan;
spIgniting:=bakspIgniting;

allPara:=bakallPara;
allGas:=bakallGas;
allWarm:=bakallWarm;
allEce:=bakallEce;
hourPara:=bakhourPara;
hourGas:=bakhourGas;
hourWarm:=bakhourWarm;
hourEce:=bakhourEce;

Ke0001:=bakKe0001;
Ke0002:=bakKe0002;
Ke0003:=bakKe0003;
Ke0004:=bakKe0004;
Ke0005:=bakKe0005;

Kmix001:=bakKmix001;
Kmix002:=bakKmix002;
Kmix003:=bakKmix003;
Kmix004:=bakKmix004;
Kmix005:=bakKmix005;
Omix001:=bakOmix001;
Omix002:=bakOmix002;
Omix003:=bakOmix003;
Omix004:=bakOmix004;
Omix005:=bakOmix005;


Sp0008:=bakSp0008;
Sp0009:=bakSp0009;
(*Sp0010:=bakSp0010;*)

Kp0008:=bakKp0008;
Ti0008:=bakTi0008;
Td0008:=bakTd0008;
Xmin0008:=bakXmin0008;
Xmax0008:=bakXmax0008;
startSP0002:=bakstartSP0002;
ignSP0002:=bakignSP0002;
		
	END_IF;
END_IF;

firstStep:=FALSE;
backup:=1;

IF Run THEN

bakfA000:=fA000;
bakfA001:=fA001;
bakfA002:=fA002;
bakfA003:=fA003;
bakfA004:=fA004;
bakfA005:=fA005;
bakfA006:=fA006;
bakfA007:=fA007;
bakfA010:=fA010;
bakfA011:=fA011;
bakfA012:=fA012;
bakfA013:=fA013;
bakfA014:=fA014;
bakfA015:=fA015;
bakfA016:=fA016;
bakfA017:=fA017;
bakfA020:=fA020;
bakfA021:=fA021;
bakfA022:=fA022;
bakfA023:=fA023;
bakfA024:=fA024;
bakfA025:=fA025;
bakfA026:=fA026;
bakfA027:=fA027;
bakmodeGas:=modeGas;

bakSp0001:=Sp0001;
bakKp0001:=Kp0001;
bakTi0001:=Ti0001;
bakTd0001:=Td0001;
bakXmin0001:=Xmin0001;
bakXmax0001:=Xmax0001;
bakSp0002:=Sp0002;
bakKp0002:=Kp0002;
bakTi0002:=Ti0002;
bakTd0002:=Td0002;
bakXmin0002:=Xmin0002;
bakXmax0002:=Xmax0002;
bakSp0003:=Sp0003;
bakKp0003:=Kp0003;
bakTi0003:=Ti0003;
bakTd0003:=Td0003;
bakXmin0003:=Xmin0003;
bakXmax0003:=Xmax0003;
bakSp0004:=Sp0004;
bakKp0004:=Kp0004;
bakTi0004:=Ti0004;
bakTd0004:=Td0004;
bakXmin0004:=Xmin0004;
bakXmax0004:=Xmax0004;
bakSp0005:=Sp0005;
bakKp0005:=Kp0005;
bakTi0005:=Ti0005;
bakTd0005:=Td0005;
bakXmin0005:=Xmin0005;
bakXmax0005:=Xmax0005;
bakSp0006:=Sp0006;
bakKp0006:=Kp0006;
bakTi0006:=Ti0006;
bakTd0006:=Td0006;
bakXmin0006:=Xmin0006;
bakXmax0006:=Xmax0006;
bakSp0007:=Sp0007;
bakKp0007:=Kp0007;
bakTi0007:=Ti0007;
bakTd0007:=Td0007;
bakXmin0007:=Xmin0007;
bakXmax0007:=Xmax0007;
baktMeoTerm:=tMeoTerm;
baktMeoGas:=tMeoGas;
bakdGas:=dGas;
bakdTerm:=dTerm;
bakdSupp:=dSupport;
bakmaxS1:=maxS1;
bakmaxS2:=maxS2;
bakmaxS3:=maxS3;
bakmaxS4:=maxS4;
bakmaxS5:=maxS5;
bakK2001:=K2001;
bakstartPump:=startPump;
bakstartFan:=startFan;
bakstartExh:=startExh;
bakstartGas:=startGas;
bakstartTerm:=startTerm;
bakgOffset:=gOffset;
bakgGain:=gGain;
bakheatingGas:=heatingGas;
baksca_Ppara:=sca_Ppara;
bakmax_Ppara:=max_Ppara;
baksca_Tpar:=sca_Tpar;
bakmax_Tpar:=max_Tpar;
baksca_Tv3a:=sca_Tv3a;
bakmax_Tv3a:=max_Tv3a;
baksca_Fgas:=sca_Fgas;
bakmax_Fgas:=max_Fgas;
baksca_Fpara:=sca_Fpara;
bakmax_Fpara:=max_Fpara;
bakqgas:=qgas;
baksca_Fwater:=sca_Fwater;
bakmax_Fwater:=max_Fwater;
bakgTermOffset:=gTermOffset;
bakgTermGain:=gTermGain;
bakgSuppOffset:=gSuppOffset;
bakgSuppGain:=gSuppGain;

bakTpr0001:=Tpr0001;
bakTpr0002:=Tpr0002;
bakTpr0003:=Tpr0003;
bakTpr0004:=Tpr0004;
bakTpr0005:=Tpr0005;
bakTpr0006:=Tpr0006;
bakTpr0007:=Tpr0007;
bakTpr0008:=Tpr0008;
bakTpr0009:=Tpr0009;
bakTpr0010:=Tpr0010;
bakTpr0011:=Tpr0011;
bakTpr0012:=Tpr0012;
bakspTstart:=spTstart;
bakspTVentPre:=spTVentPre;
bakspTVentPost:=spTVentPost;
bakspTBlowing:=spTBlowing;
bakspStartfeed:=spStartfeed;
bakspStartExh:=spStartExh;
bakspStartfan:=spStartfan;
bakspIgniting:=spIgniting;

bakallPara:=allPara;
bakallGas:=allGas;
bakallWarm:=allWarm;
bakallEce:=allEce;
bakhourPara:=hourPara;
bakhourGas:=hourGas;
bakhourWarm:=hourWarm;
bakhourEce:=hourEce;
	
bakKe0001:=Ke0001;
bakKe0002:=Ke0002;
bakKe0003:=Ke0003;
bakKe0004:=Ke0004;
bakKe0005:=Ke0005;


bakKmix001:=Kmix001;
bakKmix002:=Kmix002;
bakKmix003:=Kmix003;
bakKmix004:=Kmix004;
bakKmix005:=Kmix005;
bakOmix001:=Omix001;
bakOmix002:=Omix002;
bakOmix003:=Omix003;
bakOmix004:=Omix004;
bakOmix005:=Omix005;

bakSp0008:=Sp0008;
bakSp0009:=Sp0009;
(*bakSp0010:=Sp0010;*)

bakKp0008:=Kp0008;
bakTi0008:=Ti0008;
bakTd0008:=Td0008;
bakXmin0008:=Xmin0008;
bakXmax0008:=Xmax0008;
bakstartSP0002:=startSP0002;

bakignSP0002:=ignSP0002;


END_IF;

Run:=FALSE;

END_PROGRAM

// MyController/Application/Prog/service
PROGRAM service
VAR
	fe_amGas: F_TRIG;
	fe_amTerm: F_TRIG;
	fe_amSupport: F_TRIG;
	
	tmp: TIME;
	
END_VAR


(*робота з регуляторами безударний перехід в ручний режим *)
IF AM001 AND xPumpAuto THEN
	cPump:=Xt0001;
END_IF;

IF AM002 AND xFanAuto AND NOT regO2en THEN
	Xt0006:=Xt0002;
	cFan:=Xt0006;
END_IF;

IF AM002 AND xFanAuto  AND regO2en THEN
	cFan:=Xt0006;
END_IF;

IF AM003 AND xExhAuto THEN
	cExh:=Xt0003;
END_IF;

IF AM005 AND xTermAuto THEN
	cTerm:=Xt0005;
END_IF;

(*Звязане управління мео температури і підпору*)
IF AmTerm AND amSupp THEN
		cSupport:=4000.0-cTerm; (*клапан підпору працює в противофазі із клапаном температури*)
END_IF;

IF AM008 THEN (*якщо включено регулятор прогріву котла*)
	cGas:=Xt0008;
END_IF;

IF AM004 AND xGasAuto THEN
	CASE modeGas OF
		0: (*регулятор тиску*)
			cGas:=Xt0004;
		1: (*регулятор витрати*)
			cGas:=Xt0007;
	END_CASE;
END_IF;



Out1:=REAL_TO_INT(cPump);
Out2:=REAL_TO_INT(cFan);
Out3:=REAL_TO_INT(cExh);
Out4:=REAL_TO_INT(cGas);

(*-----------------------------------------------------------------------------------------------------------------------------------------------------------*)
(*Робота з МЕО*)
(*Газ*)
(*Взагалі-то вся ця хрінь проситься зробити блоком але як тоді в ручну управляти виходами ? треба подумати*)

IF yGasOpen OR yGasClose THEN (*Розрахунок таймера для захисту*)
	tmp:=REAL_TO_TIME(ABS(gGas-cGas)*tMeoGas)+t#1s;
	IF tmp>tMeo1 THEN
		tMeo1:=tmp;
	END_IF
ELSE
	tMeo1:=T#1S;
END_IF

IF amGas AND NOT AM004 THEN
	IF gGas>cGas+dGas THEN (*якщо відкрито більше ніж треба*)
		yGasClose:=TRUE; (*відкрити*)
	END_IF;
	IF gGas<cGas-dGas THEN (*як закрито більше ніж треба*)
		yGasOpen:=TRUE;
	END_IF;
	IF gGas<cGas+dGas THEN
		yGasClose:=FALSE;
	END_IF;
	IF gGas>cGas-dGas THEN 
		yGasOpen:=FALSE;
	END_IF;
END_IF;

IF AM004 THEN (*все тут класно окрім того що цей регулятор дивиться виключно за тиском, без поправки на витрату а це погано*) 
	yGasOpen:=p4GasOpen AND gGas<Xmax0004; (*+ обмеження на мінімум-максимум*)
	yGasClose:=p4GasClose AND gGas>Xmin0004;
END_IF;

(*при переході в ручний режим виключити виходи, якщов включені*)
fe_amGas(CLK:=amGas);
IF fe_amGas.Q OR NOT  xGasAuto THEN
	yGasOpen:=FALSE;
	yGasClose:=FALSE;
END_IF;

(*Температура*)
IF yTermOpen OR yTermClose THEN (*Розрахунок таймера для захисту*)
	tmp:=REAL_TO_TIME(ABS(gTerm-cTerm)*tMeoTerm)+T#1S;
	IF tmp>tMeo2 THEN
		tMeo2:=tmp;
	END_IF
ELSE
	tMeo2:=T#1S;
END_IF


IF amTerm THEN
	IF gTerm>cTerm+dTerm THEN (*якщо відкрито більге ніж треба*)
		yTermClose:=TRUE; (*відкрити*)
	END_IF;
	IF gTerm<cTerm-dTerm THEN (*як закрито більше ніж треба*)
		yTermOpen:=TRUE;
	END_IF;
	IF gTerm<cTerm THEN
		yTermClose:=FALSE;
	END_IF;
	IF gTerm>cTerm THEN 
		yTermOpen:=FALSE;
	END_IF;
END_IF;
(*при переході в ручний режим виключити виходи, якщов включені*)
fe_amTerm(CLK:=amTerm);
IF fe_amTerm.Q  OR NOT xTermAuto THEN
	yTermOpen:=FALSE;
	yTermClose:=FALSE;
END_IF;

(*підпір*)
IF ySuppOpen OR ySuppClose THEN (*Розрахунок таймера для захисту*)
	tmp:=REAL_TO_TIME(ABS(gSupp-cSupport)*tMeoTerm)+T#1S;
	IF tmp>tMeo3 THEN
		tMeo3:=tmp;
	END_IF
ELSE
	tMeo3:=T#1S;
END_IF

IF amSupp  THEN
	IF gSupp>cSupport+dSupport THEN (*якщо відкрито більге ніж треба*)
		ySuppClose:=TRUE; (*відкрити*)
	END_IF;
	IF gSupp<cSupport-dSupport THEN (*як закрито більше ніж треба*)
		ySuppOpen:=TRUE;
	END_IF;
	IF gSupp<cSupport THEN
		ySuppClose:=FALSE;
	END_IF;
	IF gSupp>cSupport THEN 
		ySuppOpen:=FALSE;
	END_IF;
END_IF;
(*при переході в ручний режим виключити виходи, якщов включені*)
fe_amSupport(CLK:=amSupp);
IF fe_amSupport.Q OR NOT xTermAuto  THEN
	ySuppOpen:=FALSE;
	ySuppClose:=FALSE;
END_IF;
(*----------------------------------------------------------------------------------------------------------------------------------*)
(*Робота з ЧП*)

(*Робота із змінними MODBUS*)
linkPump:=drvPump.byCommError=0;
linkFan:=drvFan.byCommError=0;
linkExh:=drvExh.byCommError=0;
linkPD150:=PD150.byCommError=0;

(*перерахунок значень з частотників*)
PumpSpeed:=pump0*5;
PumpCurrent:=pump1*2;
PumpVoltage:=pump6*10;
PumpDC:=pump4*5;

xPumpRun:=pumpRun;

FanSpeed:=fan0*0.5; 
FanCurrent:=fan1*0.2;
FanVoltage:=fan2;
FanDC:=fan7*0.5; 
xFanRun:=fanStatus.0;

ExhSpeed:=exh0*0.5;
ExhCurrent:=exh3*2;
ExhVoltage:=exh2*10;
ExhDC:=exh10*0.5;
xExhRun:=exhStatus=1;

(* Тиск газу перед пальником *)
Pack_hi:=pdi1;
Pack_lo:=pdi2;
Pg15a:=Pack_v*40.0;


(*це для безударного переходу на автоматичний режим*)
IF NOT xPumpAuto THEN
	yStartPump:=xPumpRun; (*в ручному режимі дублювати сигнал run з чп*)
	IF linkPump AND xPumpRun THEN (*Якщо є звёязок по мережі *) 
		cPump:=PumpSpeed*1.6; (*це для безударного переходу в автомат*)
	END_IF;
END_IF;

IF NOT xFanAuto THEN
	yStartFan:=xFanRun; (*в ручному режимі дублювати сигнал run з чп*)
	IF linkFan AND xFanRun THEN (*Якщо є звёязок по мережі *) 
		cFan:=FanSpeed*1.6; (*це для безударного переходу в автомат*)
	END_IF;
END_IF;

IF NOT xExhAuto THEN (* якщо немає автомати але є сигнал робота із частотника *)
	yStartFan:=xExhRun OR  xFanRun  ; (*в ручному режимі дублювати сигнал run з чп*)
	IF linkExh AND xExhRun THEN (*Якщо є звёязок по мережі *) 
		cExh:=ExhSpeed*1.6; (*це для безударного переходу в автомат*)
	END_IF;
END_IF;

(*Підхват газових клапанів*)
IF NOT xGasAuto (*якщо перемикач управління газов в ручному режимі*) 
	AND xGasManOpen (*і відкриті відсічний та клапан пальника*) 
	AND xFire1 (*і при цьому є полум.я*) 
	THEN (* тоді організувати підхват*) 
	yCutofVal:=TRUE;
	yBurnerVal:=TRUE;
	YSafeVal:=FALSE;
	yLitherVal:=FALSE;	
END_IF; 
	
(*Для індикатора полум,я на панелі*)
IF xFire1 THEN
	IF yBurnerVal THEN
		flame:=2;
	ELSIF yLitherVal THEN
		flame:=1;
	ELSE
		flame:=3;
	END_IF;
ELSE
	flame:=0;
END_IF;

END_PROGRAM

// MyController/Application/Prog/main
PROGRAM main
VAR
	// таймер тесту дзвінка
	tmTestSerena: TON;
	// таймер запуску частотників вентирятора і димососа
	tmTstartFan: TON;
	tmTstartExh: TON;
	
	// таймер розпалу запальнички
	tmIgniting: TON;
	
	// час наповнення барабана
	tmStartfeed: TON;
	tmStartExh: TON;
	tmStartFan: TON;
	
	// таймер часу вентиляції топки
	tmTVentPre: TON;
	// таймер продувки газопровода		
	tmBlowing: TON;
	// перевірка State>ST_CHECKTIGHT виконується дуже барато раз
	stateCheckGE: BOOL;
	
	// таймер перевірки герметичості 
	tmCheckTight4: TON;
	// таймери перевірки герметичності на пусту
	tmCheckTight3: TON;
	// таймер набору газу для перевірки герметичності
	tmCheckTight2: TON;
	// таймер перевірки герметичності від тиском
	tmCheckTight1: TON;
	
	// таймер уявного полом,я
	tmXFire1: TON;
	// таймер реального полум,я
	tmXFire2: TON;
	(*оскільки в нас немає другого датчика полум,я робимо просто витримку часу*)
	tmFiring: TON;
	// таймер вентиляції після закінчення роботи 
	tmTVentPost: TON;
	
	allXAm: BOOL;
	closeGas: R_TRIG;
	
	SerOn: R_TRIG;
	Am1On: R_TRIG;
END_VAR

(*Таймери*)
(*Таймер перевірки серени*)
tmTestSerena(IN:=State=ST_TESTSERENA,PT:=T#2S);


(*Таймер вентиляції топки при запуску*)
tmTVentPre(IN:=State=ST_VENTILATION,PT:=DWORD_TO_TIME(spTVentPre));
pvTVentPre:=spTVentPre-TIME_TO_DWORD(tmTVentPre.ET);

(*таймер вентиляції топки при зупінці*)
tmTVentPost(IN:=State>ST_RUN,PT:=DWORD_TO_TIME(spTVentPost));
pvTVentPost:=spTVentPost-TIME_TO_DWORD(tmTVentPost.ET);

(*таймери перевірки герметичності*)
tmCheckTight3(IN:=stateTight=3,PT:=T#5S);
tmCheckTight2(IN:=stateTight=2,PT:=T#2S);
tmCheckTight1(IN:=stateTight=1,PT:=T#5S);

(*таймер продувки газопроводу*)
tmBlowing(IN:=State=ST_BLOWING,PT:=DWORD_TO_TIME(spTBlowing));
pvTBlowing:=spTBlowing-TIME_TO_DWORD(tmBlowing.ET);

tmxFire2(IN:=xFire1,PT:=T#5S); (*тут забита константа, можливо варно налаштувати*)

tmFiring(IN:=State=ST_FIRING,PT:=spFiring);
pvFiring:=TIME_TO_DWORD(spFiring-tmFiring.ET);

tmStartFeed(IN:=State=ST_STARTFEED,PT:=DWORD_TO_TIME(spStartFeed));
pvStartFeed:=spStartFeed-TIME_TO_DWORD(tmStartFeed.ET);

tmStartExh(IN:=State=ST_STARTEXH,PT:=DWORD_TO_TIME(spStartExh));
pvStartExh:=spStartExh-TIME_TO_DWORD(tmStartExh.ET);

tmStartFan(IN:=State=ST_STARTFAN,PT:=DWORD_TO_TIME(spStartFan));
pvStartFan:=spStartFan-TIME_TO_DWORD(tmStartFan.ET);

tmIgniting(IN:=State=ST_IGNITING,PT:=DWORD_TO_TIME(spIgniting));
pvIgniting:=spIgniting-TIME_TO_DWORD(tmIgniting.ET);



allXAm:=xPumpAuto AND xFanAuto AND xExhAuto AND xGasAuto AND xTermAuto;

(*Управління сереною*)
SerOn(CLK:=Halt);
IF SerOn.Q THEN
	ySerena:=TRUE;
END_IF;

IF xAlarmBn THEN
	ySerena:=FALSE;
END_IF;

pwmParam.tCyclTime:=T#100MS;
pwmParam.tPwmPeriod:=REAL_TO_TIME(Ti0004*1000.0);
pwmParam.xPwmInstUpdt:=TRUE;

(*---------------------------------------------------------------------------------------------------------------------------------------*)
(*головний цикл управління котлом*)
IF bnStop THEN (*Це тимчасовийй код для тестування*)
	IF State<ST_IGNITING THEN
		State:=ST_STOP;
	ELSE
		State:=ST_SHUTDOWN;

(* зупинити регулятор рівня але в процесі охолодження котла його треба підкачувати *)
(*можливо просто пересмикнути регулятор в ноль *)
		yStartPump:=FALSE; 
		cPump:=0.0;	
		AM001:=FALSE; 
		
	END_IF;
END_IF;

(*це потрібно для того щоб включити регулятор рівня в автомат*)
Am1On(CLK:=Pp7a>1000.0);

CASE State OF
	ST_STOP: (*стоп*)
	(*тут треба перевірити всі початкові умови і у випадку успіху перейти далі*)
	IF allXAm THEN
		State:=ST_WAIT; (*Якщо все в автоматі перейти на стадію очікування*)
(*тут треба написати умову перехода в автоматичний режим на робочому котлі*)
(*зараз прописано перехід в автоманичний режим на зупиненому котлі*)		
	(*Все закрити та виключити*)
		ySafeVal:=TRUE; (*при переході в автоматичний режим відкрити клапан безпеки*)
		yCutofVal:=FALSE;
		yBurnerVal:=FALSE;
		yLitherVal:=FALSE;
		
		cPump:=0.0;
		cFan:=0.0;
		cExh:=0.0;
		cGas:=0.0;
		cTerm:=0.0;
		allAM:=0; (*Виключити всі регулятори з автомата*)
		yStartFan:=FALSE;
		yStartPump:=FALSE;
	END_IF
	ST_WAIT: (*Очікування*)
	(* тут треба просто чекати на натискання кнопки пуск *)

		IF bnStart THEN (*коли натиснули кнопку пуск*)
			State:=ST_TESTSERENA; (*Перейти в стадію розпалу*)
			checkList:=0; (*обнулити список перевікор*)
		END_IF;
	ST_TESTSERENA: (*1. Тест двінка*)
		ySerena:=TRUE;
		IF tmTestSerena.Q THEN
			ySerena:=FALSE;
			State:=ST_STARTFEED;
						
			check1:=TRUE;
		END_IF;
		
	ST_STARTFEED:(*2. Пуск ПН — пуск насосів живлення.*)
	(*тут би треба набрати котел водою*)
	IF LDrum>SP0001*1.08 THEN (*Якщо барабан перебраний*) 
		State:=ST_FAIL; (*треба просигналізувати про необхідність злити воду*)		
	ELSE
		(*З підкачкою все складно, якщо в барабані тиск малий - воно туди само тече, якщо великий - треба пхати*)
		IF LDrum>SP0001*0.8 THEN (*якщо рівень в барабані більше ніж -20 мм тоді нормально*)
			State:=ST_STARTEXH;
			check2:=TRUE;
			yStartPump:=FALSE;
			cPump:=0;
		ELSE
			(*отут починається саме цікаве*)
			yStartPump:=TRUE; (*включити насос*)
			cPump:=Pp7a+0.5*(2000.0-Fwater); (*це типу П регулятор з П0 у вигляді тиску в барабані*)
			IF cPump<0.0 THEN 
				cPump:=0;
			END_IF;
			IF cPump>3500.0 THEN 
				cPump:=3500.0;
			END_IF;
		END_IF;
		
	END_IF;
	
	IF tmStartFeed.Q THEN (*якщо вийшов таймер запуску*)
		State:=ST_FAIL; (*аварія*)
	END_IF
	
	ST_STARTEXH:(*3. Пуск димососа.*)	
	IF xVacPl THEN (* перевірити наявніть розрідження в топці котла*)
		IF tmTstartExh.Q THEN (*після того як витримали час запуску *)			
			AM003:=TRUE; (*перевести в автомат*)
			State:=ST_CHECKTIGHT;
			check3:=TRUE;
			cTerm:=0.0; (*startTerm; відкрити задвижку охолодження пари на максимум, відповідно мео підпору закрити*)
		END_IF;
	END_IF
		
	IF tmStartexh.Q THEN (*якщо вийшов час значить щось пішло нетак*)
		State:=ST_FAIL;
	END_IF
		
(*4. Розпал.*)
	ST_CHECKTIGHT:	(*4.1 Перевірка герметичності.*)	
		check4:=TRUE;
	(*Алгоритм*)
	CASE stateTight OF				
		3: 
			IF tmCheckTight3.Q THEN
				stateTight:=2;
				check5:=TRUE;
			END_IF			
			IF xTight THEN (*помилка, відсічний клапан не тримає*)
					(*тут необхідно перервати процедуру*)
				ySafeVal:=TRUE;
				State:=ST_FAIL;
			END_IF
		2:	(*3 відкрити відсічний клапан, дочекатися поки спрацює датчик тиску*)
			IF tmCheckTight2.Q THEN (*якщо вийшов таймер а тиск в зоні безпеки не зявився*) 
				IF xTight THEN (*все нормально, пішли далі*)
					stateTight:=1;
					check6:=TRUE;
				ELSE
					State:=ST_FAIL;
				END_IF;					
			END_IF
		1: 	(*4 закрити відсічний клапан, зачекати трохи часу, перевірити що датчик тиску продовжує показувати 1*)
			IF tmCheckTight1.Q THEN
				IF xTight THEN (*якщо після витримки часу датчик показує тиск значить все справне *)
					stateTight:=0; (*перевірку герметичності виконано*)
					check7:=TRUE;
				ELSE
					State:=ST_FAIL;									
				END_IF				
			END_IF
		0:  (*перевірка пройдена*)
			State:=ST_STARTFAN; 
	END_CASE
	
	ST_STARTFAN:(*4.2 Пуск вентилятора*)
		IF xAirPl THEN (*дочекатися сигналу з датчику тиску повітря*)
			IF tmTStartFan.Q THEN
				AM002:=TRUE;
				check8:=TRUE;
				State:=ST_VENTILATION;
				SP0002:=startSP0002;
			END_IF;
		END_IF
		
	IF tmStartFan.Q THEN
		State:=ST_FAIL;
	END_IF

	ST_VENTILATION:(*4.3 Вентиляція*)		
	(*перевірити вихід регуляторів в режим і витримати заданий час*)
		IF tmTVentPre.Q THEN (*Провентилювали топку*)
			State:=ST_BLOWING; (*Перейти в стадію розпалу котла*)
			check9:=TRUE;
			SP0002:=ignSP0002; (*виставити завдання на тиск повітря на розпал*)			
		END_IF
	ST_BLOWING: (*4.4 Продувка газопроводів*)
		IF tmBlowing.Q THEN
			State:=ST_PREPARE;
			check10:=TRUE;
		END_IF
	ST_PREPARE: (*4.5 Підготовка.*)
	(*просто ще раз все перевірити*)
	IF xAirPl 
		AND xVacPl
		THEN
		State:=ST_IGNITING;
		cPump:=0.0;
	END_IF
	(*можливо тут для стабільного підпалювання  факела треба скинути оберти вентилятора і димососа*)
	ST_IGNITING: (*4.6 Підпал запальника*)
		IF tmXFire2.Q THEN (*якщо з,явилося полум,я*)
			check11:=TRUE;
			State:=ST_FIRING;
			
			cGas:=startGas; (*встановити задане положення газової заслінки*)
			cPump:=0.0; (*в наступному циклі регулятор рівня буде включено в автомат*)
		END_IF;
		IF tmIgniting.Q THEN (*якщо вийшов час а вогню немає*)
			State:=ST_FAIL; (*тоді фейл*)
		END_IF;
	ST_FIRING: (*4.7 Підпал пальника*)
		IF tmFiring.Q THEN
			State:=ST_HEATING;			
			(* cGas:=heatingGas; тут треба  б зробити щоб регулятор хоча б один раз крутнувася з цим значенням перед вмиканням AM008=true*)
			AM001:=TRUE; (*включити регулятор рівня в автомат*)
			AM006:=TRUE; (*регулятор концентрації кисню в автомат*)
			AM008:=TRUE; (*регулятор розігріву*)
			
		END_IF
	ST_HEATING: (*4.8 Прогрів*)
	(*тут би треба зробити регулятор температури топки*)
	IF Pp7a > 800.0 THEN (*не самий гарний варіант*) 
		yStartPump:=TRUE; (**)			
	END_IF;
	IF Pp7a>SP0004*0.85 THEN (*коли виросте в котлі тиск перейти в стан робота*)
		State:=ST_RUN;
		yStartPump:=TRUE; (**)
		AM008:=FALSE; (*Регулятор розігріві*)
		AM004:=TRUE;
		AM005:=TRUE;		
	END_IF
	ST_RUN: (*5. Робота*)
	(*тут має бути відпрацювання технологічної карти *)
	(*-------------------------------------------------------*)
	(*а може й ні, якщо регулятор О2 буде достатньо*)
	
(*5.1 Робота, набір потужності*)
(*5.2 Робота, підтримання потужності*)
(*5.3. Робота, зменшення потужності*)

(*6 Зупинка*)
(*6.1 Зупинка штатна*)
	ST_SHUTDOWN:
		(*тут мали б працювати всі регулятори*)
		IF tmTVentPost.Q THEN
			State:=ST_STOP;
		END_IF
		AM008:=FALSE;
		AM002:=FALSE;
		
	ST_FAIL:	(*6.2 Зупинка по аварії*)
		IF xAlarmBn THEN
			State:=ST_SHUTDOWN;
		END_IF;
			
(*
		IF tmTVentPost.Q THEN
			State:=ST_STOP;
		END_IF
*)		
		
END_CASE;
stWait:=State=ST_WAIT; (*для панеля для блокування і розблокування кнопок пуск/стоп*)

(*включити захист на повну котушку*)
IF State>ST_PREPARE AND Halt THEN (*якщо немає полум,я*)
	State:=ST_FAIL;
END_IF;

stateCheckGE:=State>ST_CHECKTIGHT;

tmTstartFan(IN:= (stateCheckGE AND yStartFan) ,PT:=DWORD_TO_TIME(spTstart));
tmTstartExh(IN:= (State>ST_STARTFEED AND yStartFan) ,PT:=DWORD_TO_TIME(spTstart));
(*таймер контролю уявного полум,я*)
tmXFire1(IN:=(xFire1 AND State>ST_WAIT AND State<ST_PREPARE),PT:=T#1S);

(*в стані ST_WAIT можна керувати виконавчими механізмами вручну*)
IF State>ST_WAIT THEN (* купа всякого різного управління в автоматичному режимі*)
	(*контроль уявного полум,я*)
	IF tmXFire1.Q THEN 
		check0:=FALSE;
		State:=ST_FAIL;
	ELSE
		check0:=TRUE;
	END_IF

	IF State<>ST_CHECKTIGHT THEN (*підготувати змінну для перевірки герметичності*)
		stateTight:=3; 
	END_IF
(*-----------------------------------------------------------------------------------------------------------------*)
	(*управління клапаном безпеки*)
	ySafeVal:=(State>ST_CHECKTIGHT AND State<ST_FIRING) OR State>ST_RUN;
	
	(*управління відсічним клапаном*)
	yCutofVal:= (State=ST_CHECKTIGHT AND stateTight=2) (*набор зони безпеки для перевірки герметичності*) 
				OR (ST_VENTILATION < State AND State < ST_SHUTDOWN);  (*робота*)
	(*управління клапаном пальника*)
	yBurnerVal:= (State>ST_IGNITING AND State<ST_SHUTDOWN); 
	(*Управління клапаном запальника*)
	yLitherVal:=ST_PREPARE < State AND State < ST_HEATING;
 
	(*управління трансформатором*)
	yIgniter:=State=ST_IGNITING AND NOT xFire1; (*подати іскру якщо стадія підпалу запальнички і вона не горить.*)
	
	(*управління мео газу*)
	(*
	IF ST_BLOWING < State AND State < ST_HEATING AND YBurnerVal THEN
		cGas:=startGas;
	END_IF
	*)
(*-----------------------------------------------------------------------------------------------------------------*)
	(*управління живильним насосом*)
	(*код звідси перенесен вище*)

	
	(*управління димососм*)
	IF State>ST_STARTFEED THEN (*як запустили живильний насос і набрали в котел води*)
		yStartFan:=TRUE; (*включити димосос і вентилятор*)
		IF NOT tmTstartExh.Q THEN (*після того як витримали час запуску *)			
			cExh:=startExh; (*вивести стартове значення*)
		END_IF;
	ELSE
		yStartFan:=FALSE; (*в іншій ситуації виключити*)
		cExh:=0.0;
	END_IF;
	
	(*управління вентилятором*)
	IF stateCheckGE AND yStartFan THEN
		IF NOT tmTStartFan.Q THEN
			cFan:=startFan;
		END_IF
	ELSE
		cFan:=0.0;
	END_IF
	

END_IF;

(*при вимиканні стейт машини управління котлом клапана газу закрити а клапан безпеки відкрити*)
closeGas(CLK:=State<ST_WAIT);
IF closeGas.Q THEN
	yCutofVal:=FALSE;
	yBurnerVal:=FALSE;
	ySafeVal:=TRUE;
END_IF

(*Скину всі натиснуті кнопки*)
bnAll:=0;

(*------------------------------*)

END_PROGRAM

// MyController/Application/Prog/SafeTmr
PROGRAM SafeTmr
VAR
	tonMeo1: TON;
	tonMeo2: TON;
	tonMeo3: TON;
	rsMeo1: RS;
	rsMeo2: RS;
	rsMeo3: RS;

	tonAl1: TON;
	tonAl2: TON;
	tonAl3: TON;
	tonAl4: TON;
	tonAl5: TON;
	tonAl6: TON;
	tonAl7: TON;
	tonAl8: TON;
	tonAl9: TON;
	tonAl10: TON;
	tonAl11: TON;

	rsAl1: RS;
	rsAl2: RS;
	rsAl3: RS;
	rsAl4: RS;
	rsAl5: RS;
	rsAl6: RS;
	rsAl7: RS;
	rsAl8: RS;
	rsAl9: RS;
	rsAl10: RS;
	rsAl11: RS;

	tonMeo1d: TIME;
	alarmCV: R_TRIG;
	alarmReset: BOOL;
	blink0: Util.BLINK;

	TON_0: TON;
	enT: BOOL;
	ptT: TIME;
	etT: TIME;
	qT: BOOL;
END_VAR
VAR // added by the converter: edge detectors and wires of the graphical bodies
    _w1 : BOOL;
    _rt1, _rt2, _rt3, _rt4, _rt5, _rt6, _rt7, _rt8 : R_TRIG;
END_VAR

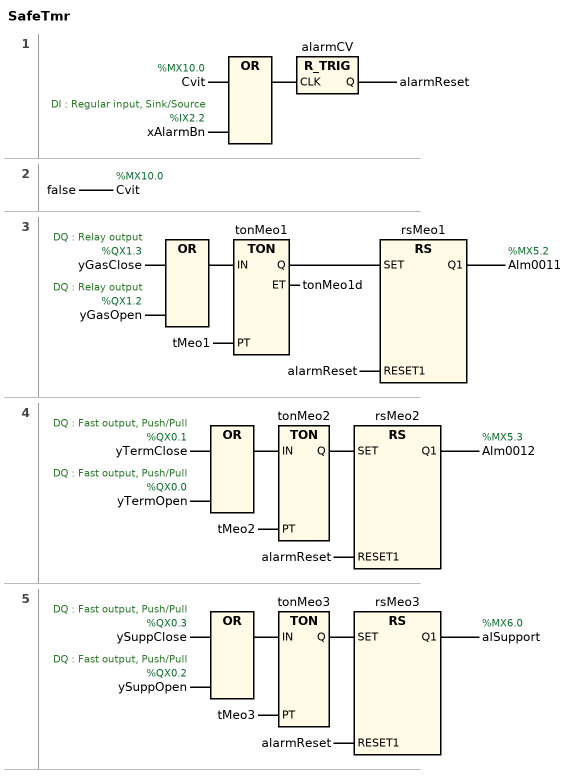
// NETWORK 1
//   Cvit: AT %MX10.0
//   xAlarmBn: DI : Regular input, Sink/Source | AT %IX2.2
alarmCV(CLK := Cvit OR xAlarmBn); // R_TRIG
alarmReset := alarmCV.Q;

// NETWORK 2
//   Cvit: AT %MX10.0
Cvit := false;

// NETWORK 3
//   yGasClose: DQ : Relay output | AT %QX1.3
//   yGasOpen: DQ : Relay output | AT %QX1.2
//   Alm0011: AT %MX5.2
tonMeo1(IN := yGasClose OR yGasOpen, PT := tMeo1, ET => tonMeo1d); // TON
rsMeo1(SET := tonMeo1.Q, RESET1 := alarmReset); // RS
Alm0011 := rsMeo1.Q1;

// NETWORK 4
//   yTermClose: DQ : Fast output, Push/Pull | AT %QX0.1
//   yTermOpen: DQ : Fast output, Push/Pull | AT %QX0.0
//   Alm0012: AT %MX5.3
tonMeo2(IN := yTermClose OR yTermOpen, PT := tMeo2); // TON
rsMeo2(SET := tonMeo2.Q, RESET1 := alarmReset); // RS
Alm0012 := rsMeo2.Q1;

// NETWORK 5
//   ySuppClose: DQ : Fast output, Push/Pull | AT %QX0.3
//   ySuppOpen: DQ : Fast output, Push/Pull | AT %QX0.2
//   alSupport: AT %MX6.0
tonMeo3(IN := ySuppClose OR ySuppOpen, PT := tMeo3); // TON
rsMeo3(SET := tonMeo3.Q, RESET1 := alarmReset); // RS
alSupport := rsMeo3.Q1;

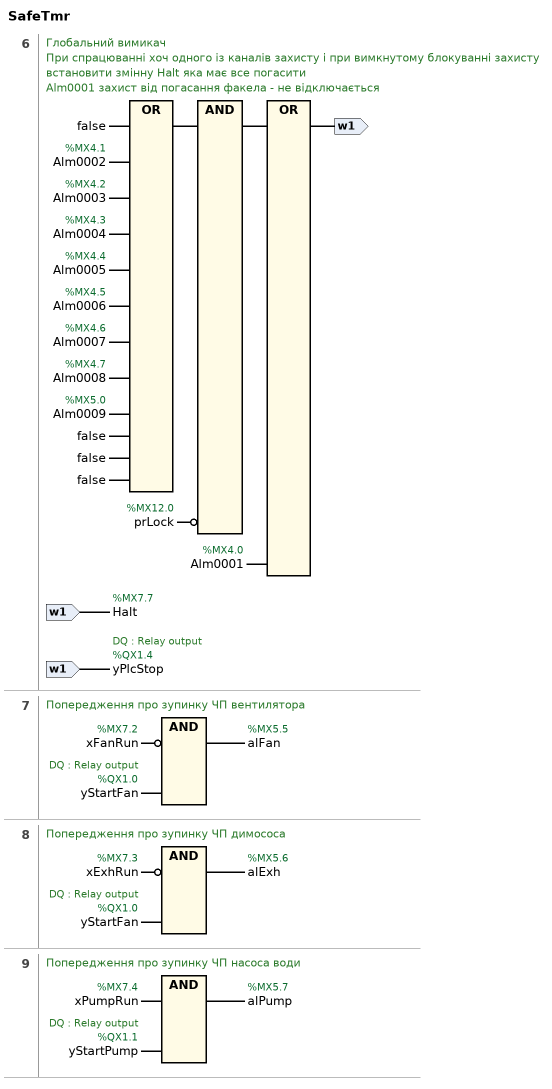
// NETWORK 6
// Глобальний вимикач
// При спрацюванні хоч одного із каналів захисту і при вимкнутому блокуванні захисту
// встановити змінну Halt яка має все погасити
// Alm0001 захист від погасання факела - не відключається
//   Alm0002: AT %MX4.1
//   Alm0003: AT %MX4.2
//   Alm0004: AT %MX4.3
//   Alm0005: AT %MX4.4
//   Alm0006: AT %MX4.5
//   Alm0007: AT %MX4.6
//   Alm0008: AT %MX4.7
//   Alm0009: AT %MX5.0
//   prLock: AT %MX12.0
//   Alm0001: AT %MX4.0
//   Halt: AT %MX7.7
//   yPlcStop: DQ : Relay output | AT %QX1.4
_w1 := (false OR Alm0002 OR Alm0003 OR Alm0004 OR Alm0005 OR Alm0006 OR Alm0007 OR Alm0008 OR Alm0009 OR false OR false OR false) AND NOT prLock OR Alm0001;
Halt := _w1;
yPlcStop := _w1;

// NETWORK 7
// Попередження про зупинку ЧП вентилятора
//   xFanRun: AT %MX7.2
//   yStartFan: DQ : Relay output | AT %QX1.0
//   alFan: AT %MX5.5
alFan := NOT xFanRun AND yStartFan;

// NETWORK 8
// Попередження про зупинку ЧП димососа
//   xExhRun: AT %MX7.3
//   yStartFan: DQ : Relay output | AT %QX1.0
//   alExh: AT %MX5.6
alExh := NOT xExhRun AND yStartFan;

// NETWORK 9
// Попередження про зупинку ЧП насоса води
//   xPumpRun: AT %MX7.4
//   yStartPump: DQ : Relay output | AT %QX1.1
//   alPump: AT %MX5.7
alPump := xPumpRun AND yStartPump;

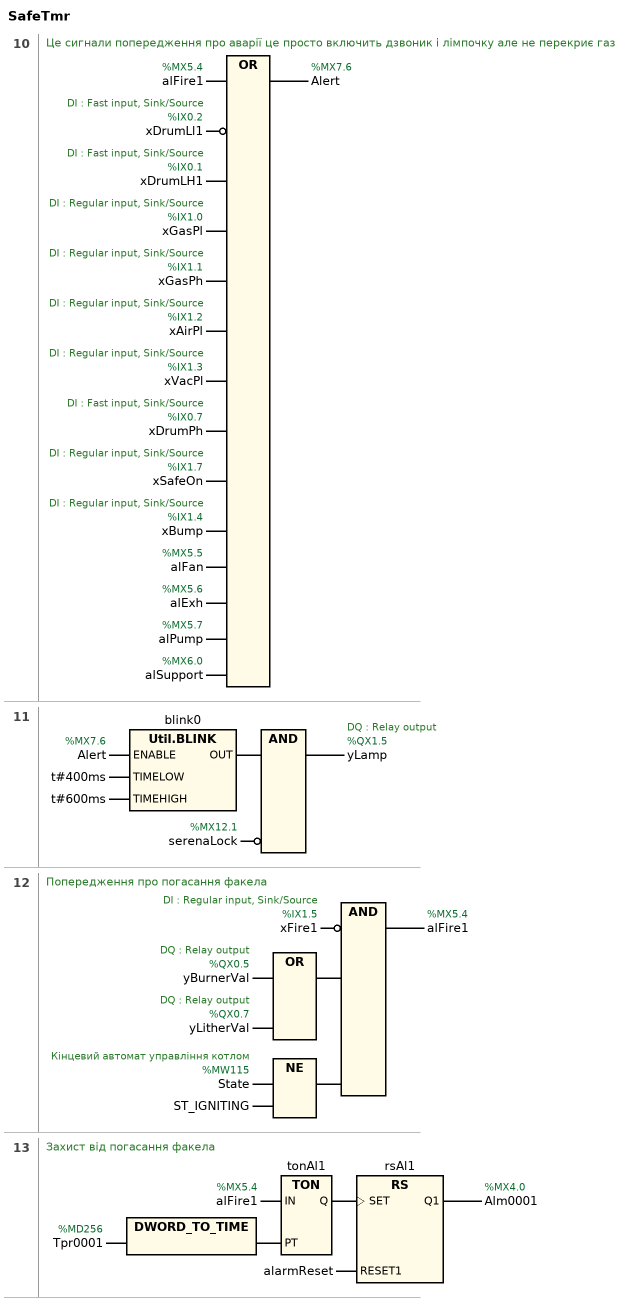
// NETWORK 10
// Це сигнали попередження про аварії це просто включить дзвоник і лімпочку але не перекриє газ
//   alFire1: AT %MX5.4
//   xDrumLl1: DI : Fast input, Sink/Source | AT %IX0.2
//   xDrumLH1: DI : Fast input, Sink/Source | AT %IX0.1
//   xGasPl: DI : Regular input, Sink/Source | AT %IX1.0
//   xGasPh: DI : Regular input, Sink/Source | AT %IX1.1
//   xAirPl: DI : Regular input, Sink/Source | AT %IX1.2
//   xVacPl: DI : Regular input, Sink/Source | AT %IX1.3
//   xDrumPh: DI : Fast input, Sink/Source | AT %IX0.7
//   xSafeOn: DI : Regular input, Sink/Source | AT %IX1.7
//   xBump: DI : Regular input, Sink/Source | AT %IX1.4
//   alFan: AT %MX5.5
//   alExh: AT %MX5.6
//   alPump: AT %MX5.7
//   alSupport: AT %MX6.0
//   Alert: AT %MX7.6
Alert := alFire1 OR NOT xDrumLl1 OR xDrumLH1 OR xGasPl OR xGasPh OR xAirPl OR xVacPl OR xDrumPh OR xSafeOn OR xBump OR alFan OR alExh OR alPump OR alSupport;

// NETWORK 11
//   Alert: AT %MX7.6
//   serenaLock: AT %MX12.1
//   yLamp: DQ : Relay output | AT %QX1.5
blink0(ENABLE := Alert, TIMELOW := t#400ms, TIMEHIGH := t#600ms); // Util.BLINK
yLamp := blink0.OUT AND NOT serenaLock;

// NETWORK 12
// Попередження про погасання факела
//   xFire1: DI : Regular input, Sink/Source | AT %IX1.5
//   yBurnerVal: DQ : Relay output | AT %QX0.5
//   yLitherVal: DQ : Relay output | AT %QX0.7
//   State: Кінцевий автомат управління котлом | AT %MW115
//   alFire1: AT %MX5.4
alFire1 := NOT xFire1 AND (yBurnerVal OR yLitherVal) AND State <> ST_IGNITING;

// NETWORK 13
// Захист від погасання факела
//   alFire1: AT %MX5.4
//   Tpr0001: AT %MD256
//   Alm0001: AT %MX4.0
tonAl1(IN := alFire1, PT := DWORD_TO_TIME(Tpr0001)); // TON
_rt1(CLK := tonAl1.Q);
rsAl1(SET := _rt1.Q, RESET1 := alarmReset); // RS
Alm0001 := rsAl1.Q1;

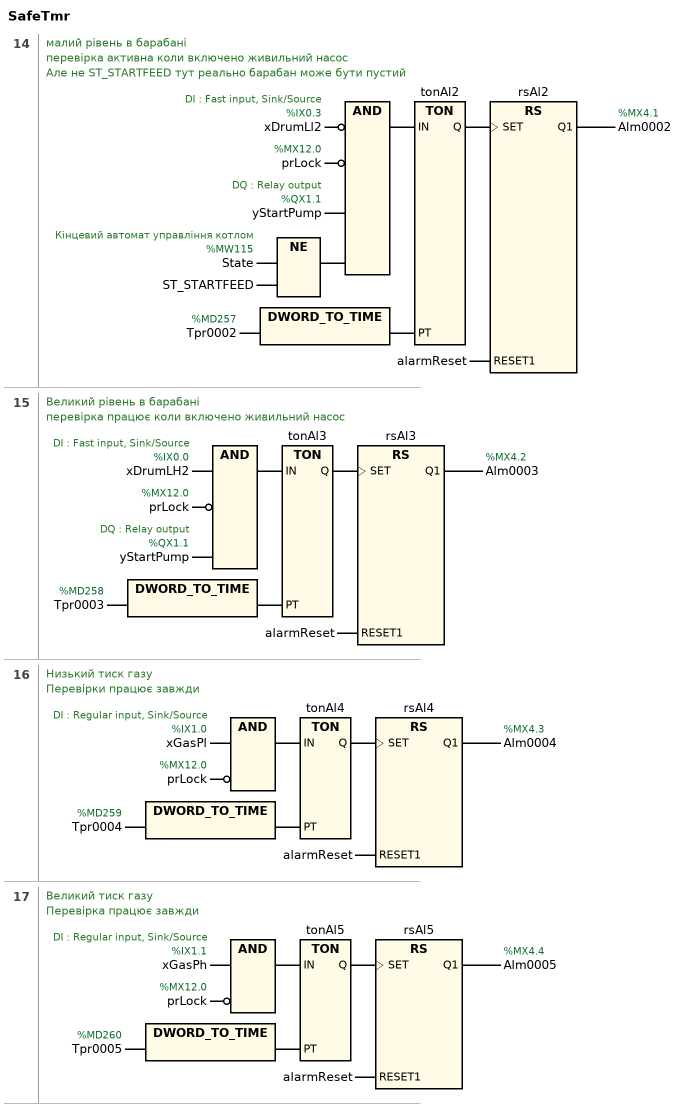
// NETWORK 14
// малий рівень в барабані
// перевірка активна коли включено живильний насос
// Але не ST_STARTFEED тут реально барабан може бути пустий
//   xDrumLl2: DI : Fast input, Sink/Source | AT %IX0.3
//   prLock: AT %MX12.0
//   yStartPump: DQ : Relay output | AT %QX1.1
//   State: Кінцевий автомат управління котлом | AT %MW115
//   Tpr0002: AT %MD257
//   Alm0002: AT %MX4.1
tonAl2(IN := NOT xDrumLl2 AND NOT prLock AND yStartPump AND State <> ST_STARTFEED, PT := DWORD_TO_TIME(Tpr0002)); // TON
_rt2(CLK := tonAl2.Q);
rsAl2(SET := _rt2.Q, RESET1 := alarmReset); // RS
Alm0002 := rsAl2.Q1;

// NETWORK 15
// Великий рівень в барабані
// перевірка працює коли включено живильний насос
//   xDrumLH2: DI : Fast input, Sink/Source | AT %IX0.0
//   prLock: AT %MX12.0
//   yStartPump: DQ : Relay output | AT %QX1.1
//   Tpr0003: AT %MD258
//   Alm0003: AT %MX4.2
tonAl3(IN := xDrumLH2 AND NOT prLock AND yStartPump, PT := DWORD_TO_TIME(Tpr0003)); // TON
_rt3(CLK := tonAl3.Q);
rsAl3(SET := _rt3.Q, RESET1 := alarmReset); // RS
Alm0003 := rsAl3.Q1;

// NETWORK 16
// Низький тиск газу
// Перевірки працює завжди
//   xGasPl: DI : Regular input, Sink/Source | AT %IX1.0
//   prLock: AT %MX12.0
//   Tpr0004: AT %MD259
//   Alm0004: AT %MX4.3
tonAl4(IN := xGasPl AND NOT prLock, PT := DWORD_TO_TIME(Tpr0004)); // TON
_rt4(CLK := tonAl4.Q);
rsAl4(SET := _rt4.Q, RESET1 := alarmReset); // RS
Alm0004 := rsAl4.Q1;

// NETWORK 17
// Великий тиск газу
// Перевірка працює завжди
//   xGasPh: DI : Regular input, Sink/Source | AT %IX1.1
//   prLock: AT %MX12.0
//   Tpr0005: AT %MD260
//   Alm0005: AT %MX4.4
tonAl5(IN := xGasPh AND NOT prLock, PT := DWORD_TO_TIME(Tpr0005)); // TON
_rt5(CLK := tonAl5.Q);
rsAl5(SET := _rt5.Q, RESET1 := alarmReset); // RS
Alm0005 := rsAl5.Q1;

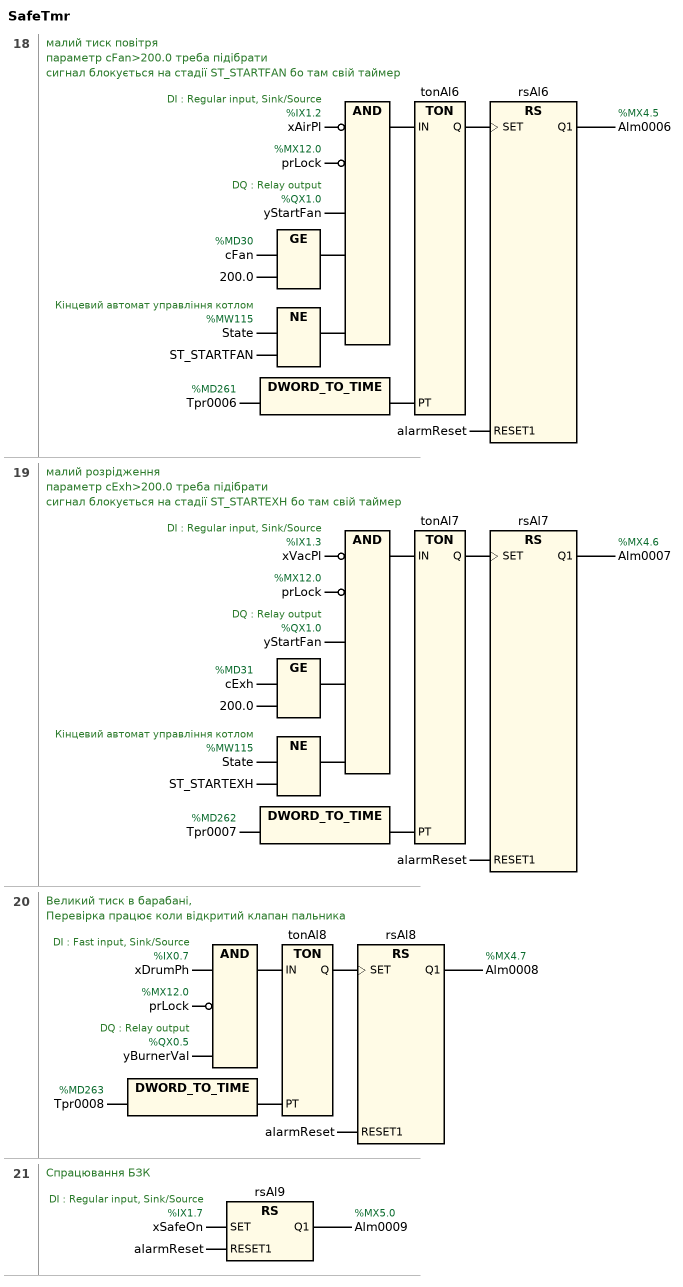
// NETWORK 18
// малий тиск повітря
// параметр cFan>200.0 треба підібрати
// сигнал блокується на стадії ST_STARTFAN бо там свій таймер
//   xAirPl: DI : Regular input, Sink/Source | AT %IX1.2
//   prLock: AT %MX12.0
//   yStartFan: DQ : Relay output | AT %QX1.0
//   cFan: AT %MD30
//   State: Кінцевий автомат управління котлом | AT %MW115
//   Tpr0006: AT %MD261
//   Alm0006: AT %MX4.5
tonAl6(IN := NOT xAirPl AND NOT prLock AND yStartFan AND cFan >= 200.0 AND State <> ST_STARTFAN, PT := DWORD_TO_TIME(Tpr0006)); // TON
_rt6(CLK := tonAl6.Q);
rsAl6(SET := _rt6.Q, RESET1 := alarmReset); // RS
Alm0006 := rsAl6.Q1;

// NETWORK 19
// малий розрідження
// параметр cExh>200.0 треба підібрати
// сигнал блокується на стадії ST_STARTEXH бо там свій таймер
//   xVacPl: DI : Regular input, Sink/Source | AT %IX1.3
//   prLock: AT %MX12.0
//   yStartFan: DQ : Relay output | AT %QX1.0
//   cExh: AT %MD31
//   State: Кінцевий автомат управління котлом | AT %MW115
//   Tpr0007: AT %MD262
//   Alm0007: AT %MX4.6
tonAl7(IN := NOT xVacPl AND NOT prLock AND yStartFan AND cExh >= 200.0 AND State <> ST_STARTEXH, PT := DWORD_TO_TIME(Tpr0007)); // TON
_rt7(CLK := tonAl7.Q);
rsAl7(SET := _rt7.Q, RESET1 := alarmReset); // RS
Alm0007 := rsAl7.Q1;

// NETWORK 20
// Великий тиск в барабані,
// Перевірка працює коли відкритий клапан пальника
//   xDrumPh: DI : Fast input, Sink/Source | AT %IX0.7
//   prLock: AT %MX12.0
//   yBurnerVal: DQ : Relay output | AT %QX0.5
//   Tpr0008: AT %MD263
//   Alm0008: AT %MX4.7
tonAl8(IN := xDrumPh AND NOT prLock AND yBurnerVal, PT := DWORD_TO_TIME(Tpr0008)); // TON
_rt8(CLK := tonAl8.Q);
rsAl8(SET := _rt8.Q, RESET1 := alarmReset); // RS
Alm0008 := rsAl8.Q1;

// NETWORK 21
// Спрацювання БЗК
//   xSafeOn: DI : Regular input, Sink/Source | AT %IX1.7
//   Alm0009: AT %MX5.0
rsAl9(SET := xSafeOn, RESET1 := alarmReset); // RS
Alm0009 := rsAl9.Q1;

END_PROGRAM

// MyController/Application/Prog/Analog
PROGRAM Analog
VAR
	AVG000: SE_TBX.Filter_MovingAverage;
	AVG001: SE_TBX.Filter_MovingAverage;
	AVG002: SE_TBX.Filter_MovingAverage;
	AVG003: SE_TBX.Filter_MovingAverage;
	AVG004: SE_TBX.Filter_MovingAverage;
	AVG005: SE_TBX.Filter_MovingAverage;
	AVG006: SE_TBX.Filter_MovingAverage;
	AVG007: SE_TBX.Filter_MovingAverage;
	AVG010: SE_TBX.Filter_MovingAverage;
	AVG011: SE_TBX.Filter_MovingAverage;
	AVG012: SE_TBX.Filter_MovingAverage;
	AVG013: SE_TBX.Filter_MovingAverage;
	AVG014: SE_TBX.Filter_MovingAverage;
	AVG015: SE_TBX.Filter_MovingAverage;
	AVG016: SE_TBX.Filter_MovingAverage;
	AVG017: SE_TBX.Filter_MovingAverage;
	AVG020: SE_TBX.Filter_MovingAverage;
	AVG021: SE_TBX.Filter_MovingAverage;
	AVG022: SE_TBX.Filter_MovingAverage;
	AVG023: SE_TBX.Filter_MovingAverage;
	AVG024: SE_TBX.Filter_MovingAverage;
	AVG025: SE_TBX.Filter_MovingAverage;
	AVG026: SE_TBX.Filter_MovingAverage;
	AVG027: SE_TBX.Filter_MovingAverage;

	Vx_int: REAL;
	
	Fpara_ob: REAL;
	LIN_TRAFO_Ter: LIN_TRAFO;
	LIN_TRAFO_Presh: LIN_TRAFO;
	parDensity: REAL;
	
END_VAR
VAR // added by the converter: edge detectors and wires of the graphical bodies
    _rt1, _rt2, _rt3, _rt4, _rt5, _rt6, _rt7, _rt8, _rt9, _rt10, _rt11, _rt12, _rt13, _rt14, _rt15, _rt16, _rt17, _rt18, _rt19, _rt20, _rt21, _rt22, _rt23, _rt24 : R_TRIG;
    _w1 : REAL;
END_VAR

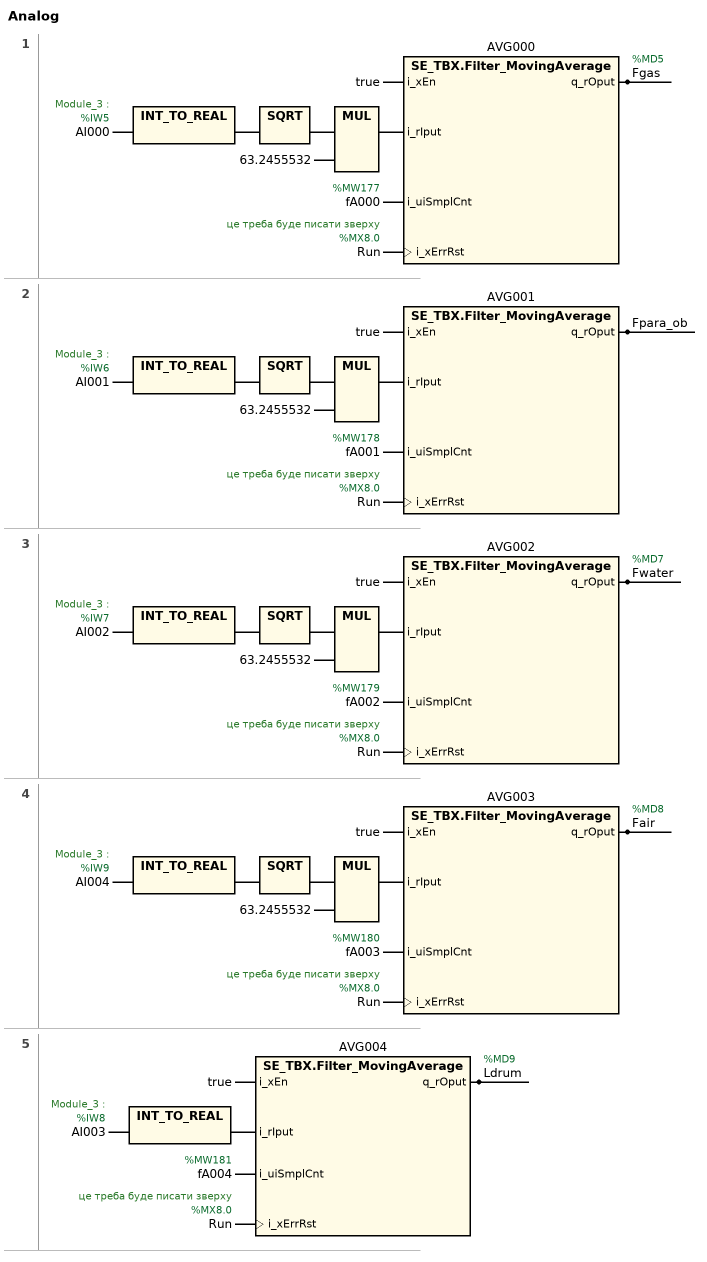
// NETWORK 1
//   AI000: Module_3 : | AT %IW5
//   fA000: AT %MW177
//   Run: це треба буде писати зверху | AT %MX8.0
//   Fgas: AT %MD5
_rt1(CLK := Run);
AVG000(
    i_xEn := true,
    i_rIput := SQRT(INT_TO_REAL(AI000)) * 63.2455532,
    i_uiSmplCnt := fA000,
    i_xErrRst := _rt1.Q,
    q_rOput => Fgas); // SE_TBX.Filter_MovingAverage

// NETWORK 2
//   AI001: Module_3 : | AT %IW6
//   fA001: AT %MW178
//   Run: це треба буде писати зверху | AT %MX8.0
_rt2(CLK := Run);
AVG001(
    i_xEn := true,
    i_rIput := SQRT(INT_TO_REAL(AI001)) * 63.2455532,
    i_uiSmplCnt := fA001,
    i_xErrRst := _rt2.Q,
    q_rOput => Fpara_ob); // SE_TBX.Filter_MovingAverage

// NETWORK 3
//   AI002: Module_3 : | AT %IW7
//   fA002: AT %MW179
//   Run: це треба буде писати зверху | AT %MX8.0
//   Fwater: AT %MD7
_rt3(CLK := Run);
AVG002(
    i_xEn := true,
    i_rIput := SQRT(INT_TO_REAL(AI002)) * 63.2455532,
    i_uiSmplCnt := fA002,
    i_xErrRst := _rt3.Q,
    q_rOput => Fwater); // SE_TBX.Filter_MovingAverage

// NETWORK 4
//   AI004: Module_3 : | AT %IW9
//   fA003: AT %MW180
//   Run: це треба буде писати зверху | AT %MX8.0
//   Fair: AT %MD8
_rt4(CLK := Run);
AVG003(
    i_xEn := true,
    i_rIput := SQRT(INT_TO_REAL(AI004)) * 63.2455532,
    i_uiSmplCnt := fA003,
    i_xErrRst := _rt4.Q,
    q_rOput => Fair); // SE_TBX.Filter_MovingAverage

// NETWORK 5
//   AI003: Module_3 : | AT %IW8
//   fA004: AT %MW181
//   Run: це треба буде писати зверху | AT %MX8.0
//   Ldrum: AT %MD9
_rt5(CLK := Run);
AVG004(
    i_xEn := true,
    i_rIput := INT_TO_REAL(AI003),
    i_uiSmplCnt := fA004,
    i_xErrRst := _rt5.Q,
    q_rOput => Ldrum); // SE_TBX.Filter_MovingAverage

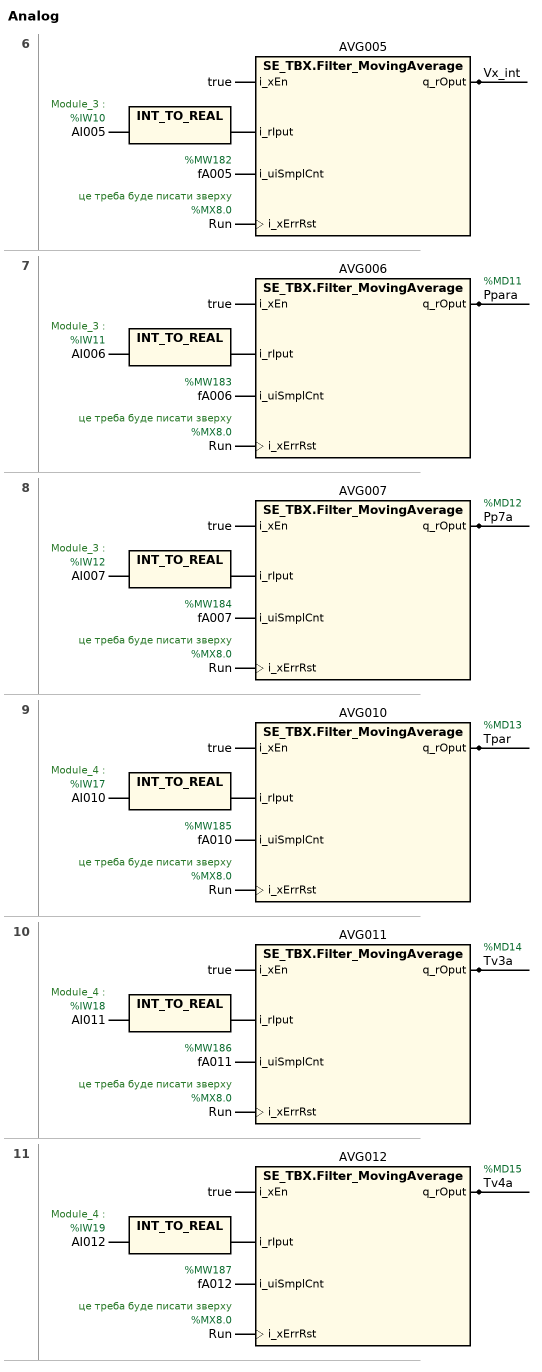
// NETWORK 6
//   AI005: Module_3 : | AT %IW10
//   fA005: AT %MW182
//   Run: це треба буде писати зверху | AT %MX8.0
_rt6(CLK := Run);
AVG005(
    i_xEn := true,
    i_rIput := INT_TO_REAL(AI005),
    i_uiSmplCnt := fA005,
    i_xErrRst := _rt6.Q,
    q_rOput => Vx_int); // SE_TBX.Filter_MovingAverage

// NETWORK 7
//   AI006: Module_3 : | AT %IW11
//   fA006: AT %MW183
//   Run: це треба буде писати зверху | AT %MX8.0
//   Ppara: AT %MD11
_rt7(CLK := Run);
AVG006(
    i_xEn := true,
    i_rIput := INT_TO_REAL(AI006),
    i_uiSmplCnt := fA006,
    i_xErrRst := _rt7.Q,
    q_rOput => Ppara); // SE_TBX.Filter_MovingAverage

// NETWORK 8
//   AI007: Module_3 : | AT %IW12
//   fA007: AT %MW184
//   Run: це треба буде писати зверху | AT %MX8.0
//   Pp7a: AT %MD12
_rt8(CLK := Run);
AVG007(
    i_xEn := true,
    i_rIput := INT_TO_REAL(AI007),
    i_uiSmplCnt := fA007,
    i_xErrRst := _rt8.Q,
    q_rOput => Pp7a); // SE_TBX.Filter_MovingAverage

// NETWORK 9
//   AI010: Module_4 : | AT %IW17
//   fA010: AT %MW185
//   Run: це треба буде писати зверху | AT %MX8.0
//   Tpar: AT %MD13
_rt9(CLK := Run);
AVG010(
    i_xEn := true,
    i_rIput := INT_TO_REAL(AI010),
    i_uiSmplCnt := fA010,
    i_xErrRst := _rt9.Q,
    q_rOput => Tpar); // SE_TBX.Filter_MovingAverage

// NETWORK 10
//   AI011: Module_4 : | AT %IW18
//   fA011: AT %MW186
//   Run: це треба буде писати зверху | AT %MX8.0
//   Tv3a: AT %MD14
_rt10(CLK := Run);
AVG011(
    i_xEn := true,
    i_rIput := INT_TO_REAL(AI011),
    i_uiSmplCnt := fA011,
    i_xErrRst := _rt10.Q,
    q_rOput => Tv3a); // SE_TBX.Filter_MovingAverage

// NETWORK 11
//   AI012: Module_4 : | AT %IW19
//   fA012: AT %MW187
//   Run: це треба буде писати зверху | AT %MX8.0
//   Tv4a: AT %MD15
_rt11(CLK := Run);
AVG012(
    i_xEn := true,
    i_rIput := INT_TO_REAL(AI012),
    i_uiSmplCnt := fA012,
    i_xErrRst := _rt11.Q,
    q_rOput => Tv4a); // SE_TBX.Filter_MovingAverage

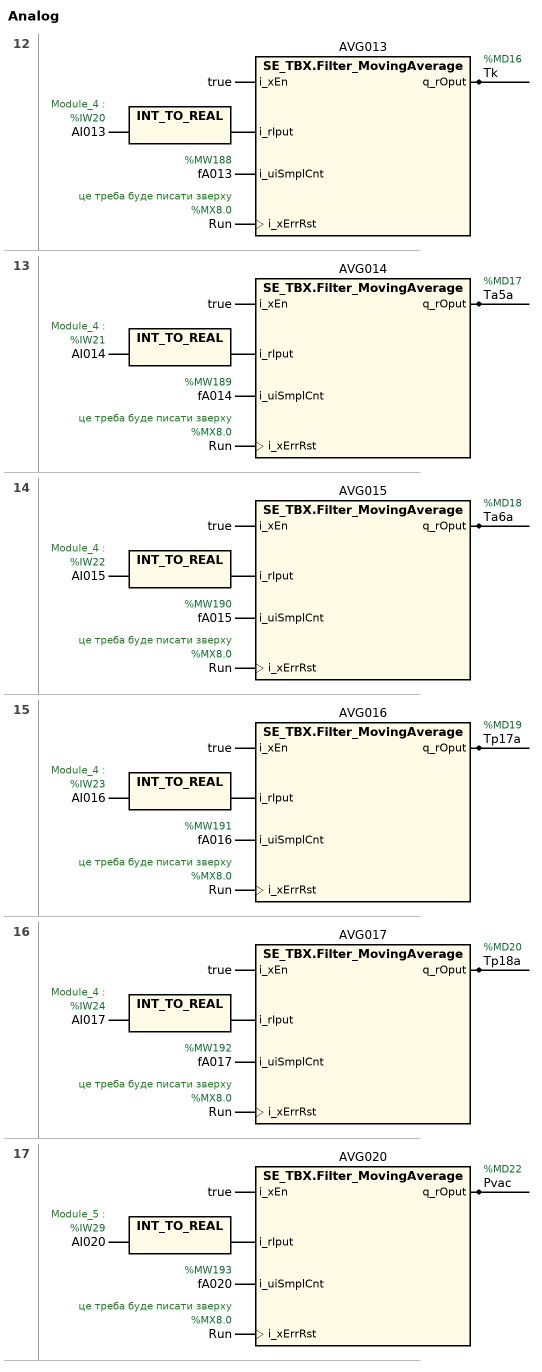
// NETWORK 12
//   AI013: Module_4 : | AT %IW20
//   fA013: AT %MW188
//   Run: це треба буде писати зверху | AT %MX8.0
//   Tk: AT %MD16
_rt12(CLK := Run);
AVG013(
    i_xEn := true,
    i_rIput := INT_TO_REAL(AI013),
    i_uiSmplCnt := fA013,
    i_xErrRst := _rt12.Q,
    q_rOput => Tk); // SE_TBX.Filter_MovingAverage

// NETWORK 13
//   AI014: Module_4 : | AT %IW21
//   fA014: AT %MW189
//   Run: це треба буде писати зверху | AT %MX8.0
//   Ta5a: AT %MD17
_rt13(CLK := Run);
AVG014(
    i_xEn := true,
    i_rIput := INT_TO_REAL(AI014),
    i_uiSmplCnt := fA014,
    i_xErrRst := _rt13.Q,
    q_rOput => Ta5a); // SE_TBX.Filter_MovingAverage

// NETWORK 14
//   AI015: Module_4 : | AT %IW22
//   fA015: AT %MW190
//   Run: це треба буде писати зверху | AT %MX8.0
//   Ta6a: AT %MD18
_rt14(CLK := Run);
AVG015(
    i_xEn := true,
    i_rIput := INT_TO_REAL(AI015),
    i_uiSmplCnt := fA015,
    i_xErrRst := _rt14.Q,
    q_rOput => Ta6a); // SE_TBX.Filter_MovingAverage

// NETWORK 15
//   AI016: Module_4 : | AT %IW23
//   fA016: AT %MW191
//   Run: це треба буде писати зверху | AT %MX8.0
//   Tp17a: AT %MD19
_rt15(CLK := Run);
AVG016(
    i_xEn := true,
    i_rIput := INT_TO_REAL(AI016),
    i_uiSmplCnt := fA016,
    i_xErrRst := _rt15.Q,
    q_rOput => Tp17a); // SE_TBX.Filter_MovingAverage

// NETWORK 16
//   AI017: Module_4 : | AT %IW24
//   fA017: AT %MW192
//   Run: це треба буде писати зверху | AT %MX8.0
//   Tp18a: AT %MD20
_rt16(CLK := Run);
AVG017(
    i_xEn := true,
    i_rIput := INT_TO_REAL(AI017),
    i_uiSmplCnt := fA017,
    i_xErrRst := _rt16.Q,
    q_rOput => Tp18a); // SE_TBX.Filter_MovingAverage

// NETWORK 17
//   AI020: Module_5 : | AT %IW29
//   fA020: AT %MW193
//   Run: це треба буде писати зверху | AT %MX8.0
//   Pvac: AT %MD22
_rt17(CLK := Run);
AVG020(
    i_xEn := true,
    i_rIput := INT_TO_REAL(AI020),
    i_uiSmplCnt := fA020,
    i_xErrRst := _rt17.Q,
    q_rOput => Pvac); // SE_TBX.Filter_MovingAverage

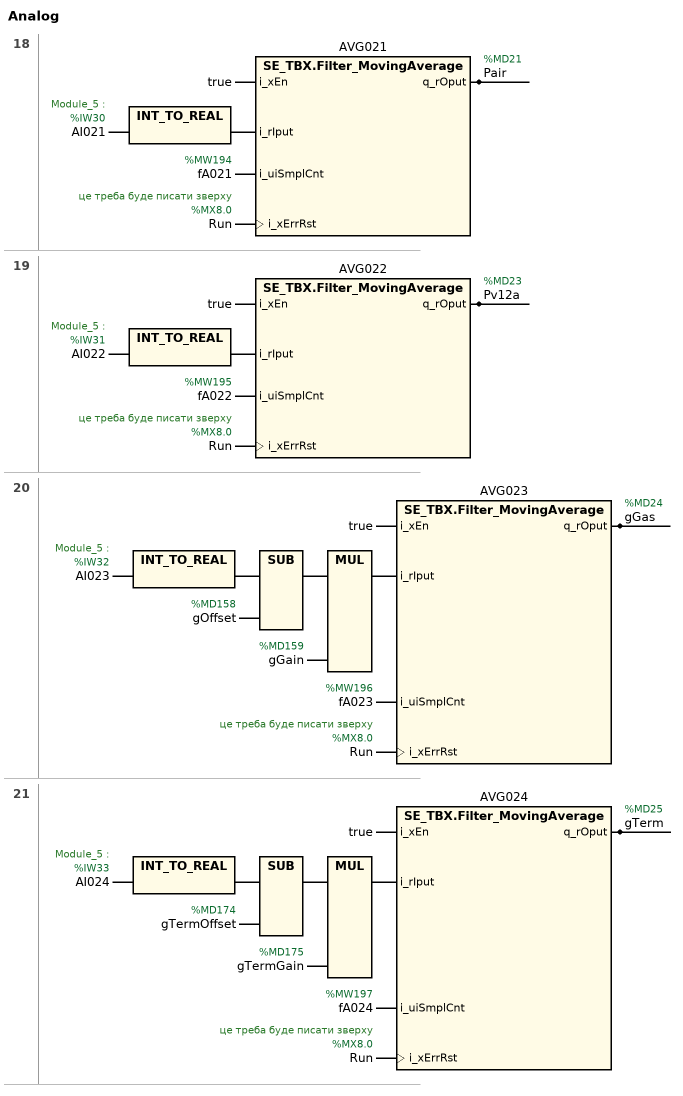
// NETWORK 18
//   AI021: Module_5 : | AT %IW30
//   fA021: AT %MW194
//   Run: це треба буде писати зверху | AT %MX8.0
//   Pair: AT %MD21
_rt18(CLK := Run);
AVG021(
    i_xEn := true,
    i_rIput := INT_TO_REAL(AI021),
    i_uiSmplCnt := fA021,
    i_xErrRst := _rt18.Q,
    q_rOput => Pair); // SE_TBX.Filter_MovingAverage

// NETWORK 19
//   AI022: Module_5 : | AT %IW31
//   fA022: AT %MW195
//   Run: це треба буде писати зверху | AT %MX8.0
//   Pv12a: AT %MD23
_rt19(CLK := Run);
AVG022(
    i_xEn := true,
    i_rIput := INT_TO_REAL(AI022),
    i_uiSmplCnt := fA022,
    i_xErrRst := _rt19.Q,
    q_rOput => Pv12a); // SE_TBX.Filter_MovingAverage

// NETWORK 20
//   AI023: Module_5 : | AT %IW32
//   gOffset: AT %MD158
//   gGain: AT %MD159
//   fA023: AT %MW196
//   Run: це треба буде писати зверху | AT %MX8.0
//   gGas: AT %MD24
_rt20(CLK := Run);
AVG023(
    i_xEn := true,
    i_rIput := (INT_TO_REAL(AI023) - gOffset) * gGain,
    i_uiSmplCnt := fA023,
    i_xErrRst := _rt20.Q,
    q_rOput => gGas); // SE_TBX.Filter_MovingAverage

// NETWORK 21
//   AI024: Module_5 : | AT %IW33
//   gTermOffset: AT %MD174
//   gTermGain: AT %MD175
//   fA024: AT %MW197
//   Run: це треба буде писати зверху | AT %MX8.0
//   gTerm: AT %MD25
_rt21(CLK := Run);
AVG024(
    i_xEn := true,
    i_rIput := (INT_TO_REAL(AI024) - gTermOffset) * gTermGain,
    i_uiSmplCnt := fA024,
    i_xErrRst := _rt21.Q,
    q_rOput => gTerm); // SE_TBX.Filter_MovingAverage

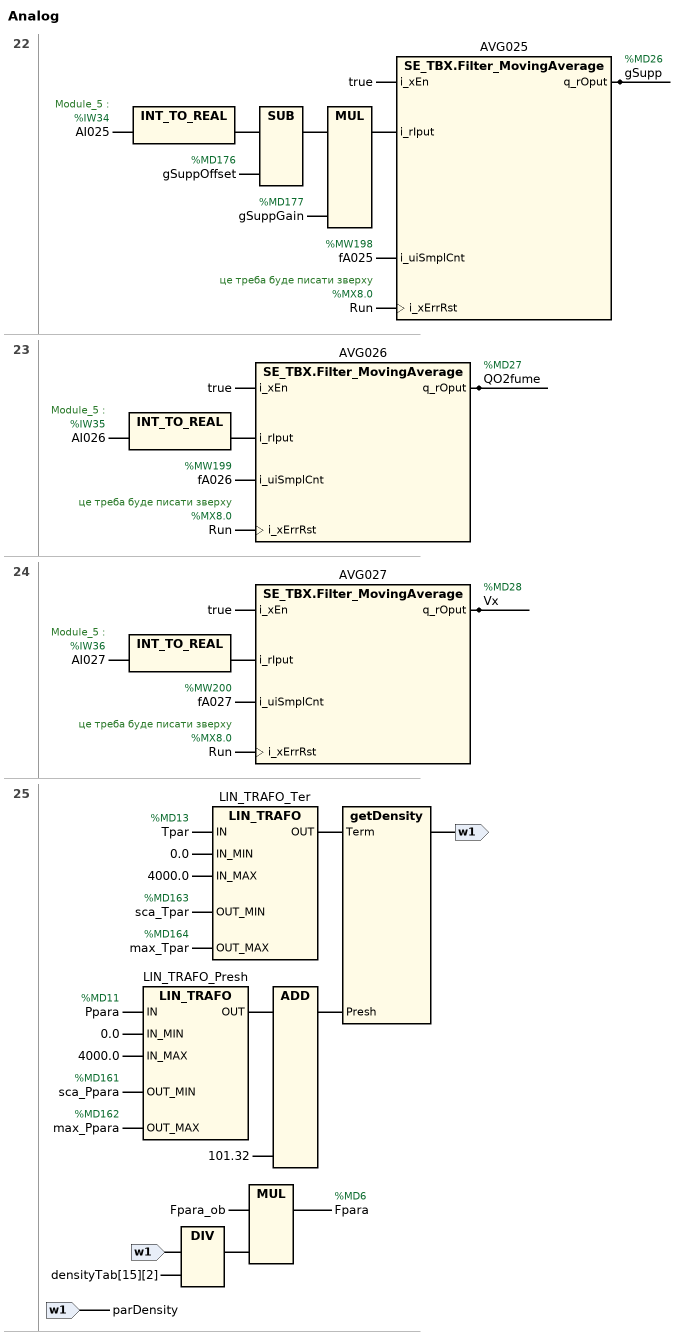
// NETWORK 22
//   AI025: Module_5 : | AT %IW34
//   gSuppOffset: AT %MD176
//   gSuppGain: AT %MD177
//   fA025: AT %MW198
//   Run: це треба буде писати зверху | AT %MX8.0
//   gSupp: AT %MD26
_rt22(CLK := Run);
AVG025(
    i_xEn := true,
    i_rIput := (INT_TO_REAL(AI025) - gSuppOffset) * gSuppGain,
    i_uiSmplCnt := fA025,
    i_xErrRst := _rt22.Q,
    q_rOput => gSupp); // SE_TBX.Filter_MovingAverage

// NETWORK 23
//   AI026: Module_5 : | AT %IW35
//   fA026: AT %MW199
//   Run: це треба буде писати зверху | AT %MX8.0
//   QO2fume: AT %MD27
_rt23(CLK := Run);
AVG026(
    i_xEn := true,
    i_rIput := INT_TO_REAL(AI026),
    i_uiSmplCnt := fA026,
    i_xErrRst := _rt23.Q,
    q_rOput => QO2fume); // SE_TBX.Filter_MovingAverage

// NETWORK 24
//   AI027: Module_5 : | AT %IW36
//   fA027: AT %MW200
//   Run: це треба буде писати зверху | AT %MX8.0
//   Vx: AT %MD28
_rt24(CLK := Run);
AVG027(
    i_xEn := true,
    i_rIput := INT_TO_REAL(AI027),
    i_uiSmplCnt := fA027,
    i_xErrRst := _rt24.Q,
    q_rOput => Vx); // SE_TBX.Filter_MovingAverage

// NETWORK 25
//   Tpar: AT %MD13
//   sca_Tpar: AT %MD163
//   max_Tpar: AT %MD164
//   Ppara: AT %MD11
//   sca_Ppara: AT %MD161
//   max_Ppara: AT %MD162
//   Fpara: AT %MD6
LIN_TRAFO_Ter(IN := Tpar, IN_MIN := 0.0, IN_MAX := 4000.0, OUT_MIN := sca_Tpar, OUT_MAX := max_Tpar); // LIN_TRAFO
LIN_TRAFO_Presh(IN := Ppara, IN_MIN := 0.0, IN_MAX := 4000.0, OUT_MIN := sca_Ppara, OUT_MAX := max_Ppara); // LIN_TRAFO
_w1 := getDensity(Term := LIN_TRAFO_Ter.OUT, Presh := LIN_TRAFO_Presh.OUT + 101.32);
Fpara := Fpara_ob * (_w1 / densityTab[15][2]);
parDensity := _w1;

END_PROGRAM

// MyController/Application/Prog/getDensity
FUNCTION getDensity : REAL
VAR_INPUT
	Term: REAL;
	Presh: REAL;
END_VAR
VAR
	ixT: INT;
	ixP: INT;
	locT: REAL;
	locP: REAL;
	
	densMin: REAL;
	densMax: REAL;
	result: REAL;
	
	err: bool;
	LIN_TRAFO_1: LIN_TRAFO;
	
END_VAR


ixT:=REAL_TO_INT(Term-200.0)/10;
IF ixT<0 THEN
	ixT:=0;
END_IF
IF ixT>29 THEN
	ixT:=29;
END_IF

locT:=Term;
IF Term<200.0 THEN
	locT:=200.0;
END_IF;
IF Term>500.0 THEN 
	locT:=500;
END_IF;


ixP:=REAL_TO_INT(Presh-1000)/500;
IF ixP<0 THEN
	ixP:=0;
END_IF

IF ixP>3 THEN
	ixP:=3;
END_IF;

locP:=Presh;
IF Presh<1000.0 THEN
	locP:=1000.0;
END_IF;
IF Presh>3000.0 THEN
	locP:=3000.0;
END_IF;

LIN_TRAFO_1( IN:= locT,IN_MIN:= termTab[ixT],IN_MAX:=termTab[ixT+1] ,OUT_MIN:= densityTab[ixT][ixP],OUT_MAX:=densityTab[ixT+1][ixP],OUT=>densMin ,ERROR=> err ); 
LIN_TRAFO_1( IN:= locT,IN_MIN:= termTab[ixT],IN_MAX:=termTab[ixT+1] ,OUT_MIN:= densityTab[ixT][ixP+1],OUT_MAX:=densityTab[ixT+1][ixP+1] ,OUT=>densMax ,ERROR=> err );
LIN_TRAFO_1( IN:= locP,IN_MIN:= preshTab[ixP],IN_MAX:=preshTab[ixP+1] ,OUT_MIN:= densMin,OUT_MAX:=densMax ,OUT=>result ,ERROR=> err );

getDensity:=result;

END_FUNCTION

// MyController/Application/Prog/control
PROGRAM control
VAR
	PID1: Util.PID;
	PID2: Util.PID;
	PID3: Util.PID;
	PID4: dualpid;
	PID5: Util.PID;
	PID6: dualpid;
	PID7: dualpid;
	PID8: Util.PID;

	DT0: Util.DERIVATIVE;
	DT1: Util.DERIVATIVE;
	DT2: Util.DERIVATIVE;
	DT3: Util.DERIVATIVE;
	DT4: Util.DERIVATIVE;
	DT5: Util.DERIVATIVE;
	der2: REAL;
	TON_0: TON;
	TON_1: TON;
	TON_2: TON;
	TON_3: TON;
	
	DER4_0: Util.DERIVATIVE;
	DER4_1: Util.DERIVATIVE;
	DER7_0: Util.DERIVATIVE;
	DER7_1: Util.DERIVATIVE;
	
	
	pid4_pwm: SE_TBX.FB_PWM;
	p4Busy: BOOL;
	p4Err: BOOL;
	
END_VAR

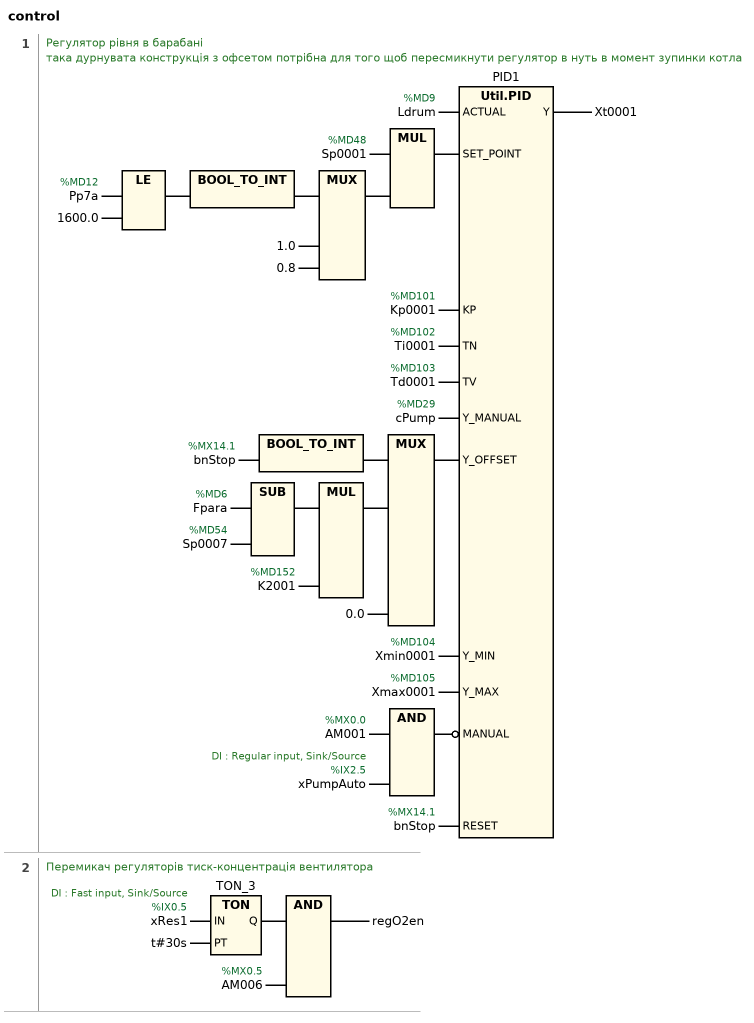
// NETWORK 1
// Регулятор рівня в барабані
// така дурнувата конструкція з офсетом потрібна для того щоб пересмикнути регулятор в нуть в момент зупинки котла
//   Ldrum: AT %MD9
//   Sp0001: AT %MD48
//   Pp7a: AT %MD12
//   Kp0001: AT %MD101
//   Ti0001: AT %MD102
//   Td0001: AT %MD103
//   cPump: AT %MD29
//   bnStop: AT %MX14.1
//   Fpara: AT %MD6
//   Sp0007: AT %MD54
//   K2001: AT %MD152
//   Xmin0001: AT %MD104
//   Xmax0001: AT %MD105
//   AM001: AT %MX0.0
//   xPumpAuto: DI : Regular input, Sink/Source | AT %IX2.5
PID1(
    ACTUAL := Ldrum,
    SET_POINT := Sp0001 * MUX(BOOL_TO_INT(Pp7a <= 1600.0), 1.0, 0.8),
    KP := Kp0001,
    TN := Ti0001,
    TV := Td0001,
    Y_MANUAL := cPump,
    Y_OFFSET := MUX(BOOL_TO_INT(bnStop), (Fpara - Sp0007) * K2001, 0.0),
    Y_MIN := Xmin0001,
    Y_MAX := Xmax0001,
    MANUAL := NOT (AM001 AND xPumpAuto),
    RESET := bnStop); // Util.PID
Xt0001 := PID1.Y;

// NETWORK 2
// Перемикач регуляторів тиск-концентрація вентилятора
//   xRes1: DI : Fast input, Sink/Source | AT %IX0.5
//   AM006: AT %MX0.5
TON_3(IN := xRes1, PT := t#30s); // TON
regO2en := TON_3.Q AND AM006;

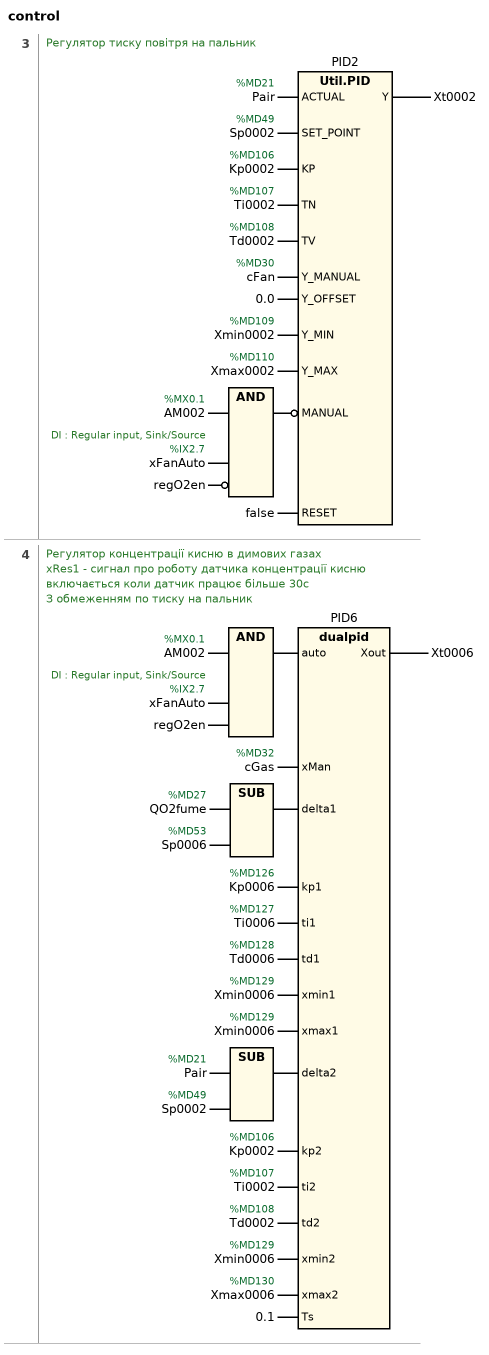
// NETWORK 3
// Регулятор тиску повітря на пальник
//   Pair: AT %MD21
//   Sp0002: AT %MD49
//   Kp0002: AT %MD106
//   Ti0002: AT %MD107
//   Td0002: AT %MD108
//   cFan: AT %MD30
//   Xmin0002: AT %MD109
//   Xmax0002: AT %MD110
//   AM002: AT %MX0.1
//   xFanAuto: DI : Regular input, Sink/Source | AT %IX2.7
PID2(
    ACTUAL := Pair,
    SET_POINT := Sp0002,
    KP := Kp0002,
    TN := Ti0002,
    TV := Td0002,
    Y_MANUAL := cFan,
    Y_OFFSET := 0.0,
    Y_MIN := Xmin0002,
    Y_MAX := Xmax0002,
    MANUAL := NOT (AM002 AND xFanAuto AND NOT regO2en),
    RESET := false); // Util.PID
Xt0002 := PID2.Y;

// NETWORK 4
// Регулятор концентрації кисню в димових газах
// xRes1 - сигнал про роботу датчика концентрації кисню
// включається коли датчик працює більше 30с
// З обмеженням по тиску на пальник
//   AM002: AT %MX0.1
//   xFanAuto: DI : Regular input, Sink/Source | AT %IX2.7
//   cGas: AT %MD32
//   QO2fume: AT %MD27
//   Sp0006: AT %MD53
//   Kp0006: AT %MD126
//   Ti0006: AT %MD127
//   Td0006: AT %MD128
//   Xmin0006: AT %MD129
//   Pair: AT %MD21
//   Sp0002: AT %MD49
//   Kp0002: AT %MD106
//   Ti0002: AT %MD107
//   Td0002: AT %MD108
//   Xmax0006: AT %MD130
PID6(
    auto := AM002 AND xFanAuto AND regO2en,
    xMan := cGas,
    delta1 := QO2fume - Sp0006,
    kp1 := Kp0006,
    ti1 := Ti0006,
    td1 := Td0006,
    xmin1 := Xmin0006,
    xmax1 := Xmin0006,
    delta2 := Pair - Sp0002,
    kp2 := Kp0002,
    ti2 := Ti0002,
    td2 := Td0002,
    xmin2 := Xmin0006,
    xmax2 := Xmax0006,
    Ts := 0.1); // dualpid
Xt0006 := PID6.Xout;

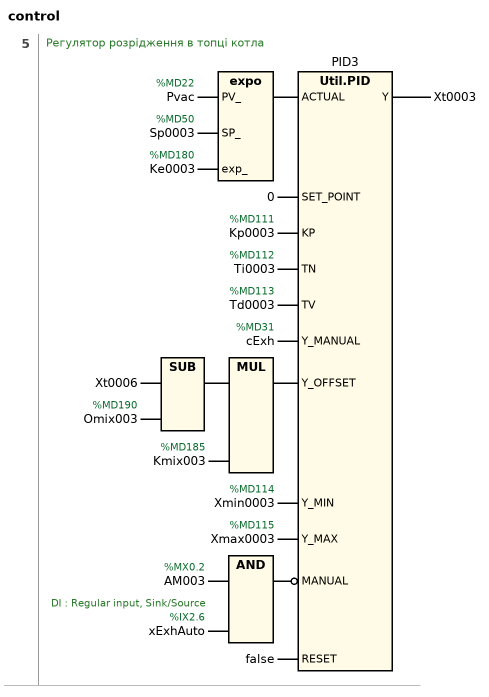
// NETWORK 5
// Регулятор розрідження в топці котла
//   Pvac: AT %MD22
//   Sp0003: AT %MD50
//   Ke0003: AT %MD180
//   Kp0003: AT %MD111
//   Ti0003: AT %MD112
//   Td0003: AT %MD113
//   cExh: AT %MD31
//   Omix003: AT %MD190
//   Kmix003: AT %MD185
//   Xmin0003: AT %MD114
//   Xmax0003: AT %MD115
//   AM003: AT %MX0.2
//   xExhAuto: DI : Regular input, Sink/Source | AT %IX2.6
PID3(
    ACTUAL := expo(PV_ := Pvac, SP_ := Sp0003, exp_ := Ke0003),
    SET_POINT := 0,
    KP := Kp0003,
    TN := Ti0003,
    TV := Td0003,
    Y_MANUAL := cExh,
    Y_OFFSET := (Xt0006 - Omix003) * Kmix003,
    Y_MIN := Xmin0003,
    Y_MAX := Xmax0003,
    MANUAL := NOT (AM003 AND xExhAuto),
    RESET := false); // Util.PID
Xt0003 := PID3.Y;

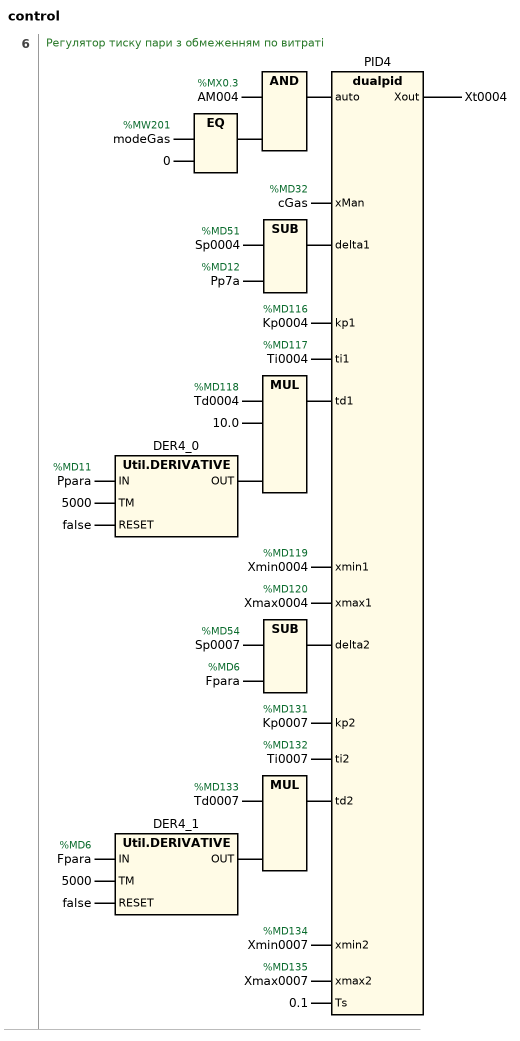
// NETWORK 6
// Регулятор тиску пари з обмеженням по витраті
//   AM004: AT %MX0.3
//   modeGas: AT %MW201
//   cGas: AT %MD32
//   Sp0004: AT %MD51
//   Pp7a: AT %MD12
//   Kp0004: AT %MD116
//   Ti0004: AT %MD117
//   Td0004: AT %MD118
//   Ppara: AT %MD11
//   Xmin0004: AT %MD119
//   Xmax0004: AT %MD120
//   Sp0007: AT %MD54
//   Fpara: AT %MD6
//   Kp0007: AT %MD131
//   Ti0007: AT %MD132
//   Td0007: AT %MD133
//   Xmin0007: AT %MD134
//   Xmax0007: AT %MD135
DER4_0(IN := Ppara, TM := 5000, RESET := false); // Util.DERIVATIVE
DER4_1(IN := Fpara, TM := 5000, RESET := false); // Util.DERIVATIVE
PID4(
    auto := AM004 AND modeGas = 0,
    xMan := cGas,
    delta1 := Sp0004 - Pp7a,
    kp1 := Kp0004,
    ti1 := Ti0004,
    td1 := Td0004 * 10.0 * DER4_0.OUT,
    xmin1 := Xmin0004,
    xmax1 := Xmax0004,
    delta2 := Sp0007 - Fpara,
    kp2 := Kp0007,
    ti2 := Ti0007,
    td2 := Td0007 * DER4_1.OUT,
    xmin2 := Xmin0007,
    xmax2 := Xmax0007,
    Ts := 0.1); // dualpid
Xt0004 := PID4.Xout;

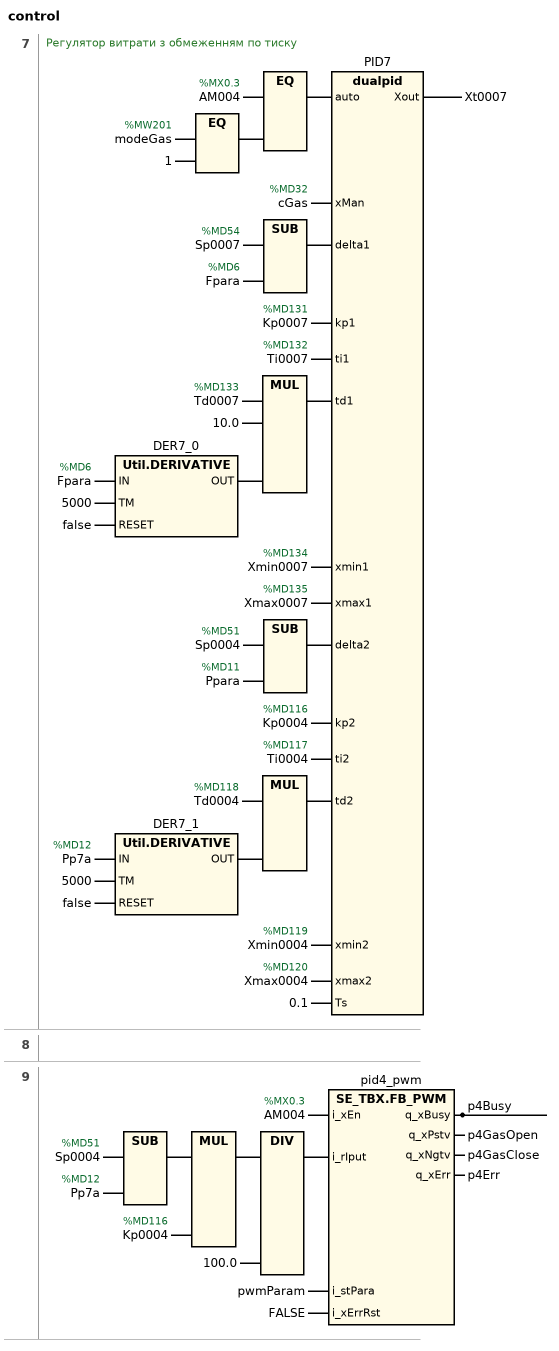
// NETWORK 7
// Регулятор витрати з обмеженням по тиску
//   AM004: AT %MX0.3
//   modeGas: AT %MW201
//   cGas: AT %MD32
//   Sp0007: AT %MD54
//   Fpara: AT %MD6
//   Kp0007: AT %MD131
//   Ti0007: AT %MD132
//   Td0007: AT %MD133
//   Xmin0007: AT %MD134
//   Xmax0007: AT %MD135
//   Sp0004: AT %MD51
//   Ppara: AT %MD11
//   Kp0004: AT %MD116
//   Ti0004: AT %MD117
//   Td0004: AT %MD118
//   Pp7a: AT %MD12
//   Xmin0004: AT %MD119
//   Xmax0004: AT %MD120
DER7_0(IN := Fpara, TM := 5000, RESET := false); // Util.DERIVATIVE
DER7_1(IN := Pp7a, TM := 5000, RESET := false); // Util.DERIVATIVE
PID7(
    auto := AM004 = (modeGas = 1),
    xMan := cGas,
    delta1 := Sp0007 - Fpara,
    kp1 := Kp0007,
    ti1 := Ti0007,
    td1 := Td0007 * 10.0 * DER7_0.OUT,
    xmin1 := Xmin0007,
    xmax1 := Xmax0007,
    delta2 := Sp0004 - Ppara,
    kp2 := Kp0004,
    ti2 := Ti0004,
    td2 := Td0004 * DER7_1.OUT,
    xmin2 := Xmin0004,
    xmax2 := Xmax0004,
    Ts := 0.1); // dualpid
Xt0007 := PID7.Xout;

// NETWORK 8

// NETWORK 9
//   AM004: AT %MX0.3
//   Sp0004: AT %MD51
//   Pp7a: AT %MD12
//   Kp0004: AT %MD116
pid4_pwm(
    i_xEn := AM004,
    i_rIput := ((Sp0004 - Pp7a) * Kp0004) / 100.0,
    i_stPara := pwmParam,
    i_xErrRst := FALSE,
    q_xBusy => p4Busy,
    q_xPstv => p4GasOpen,
    q_xNgtv => p4GasClose,
    q_xErr => p4Err); // SE_TBX.FB_PWM

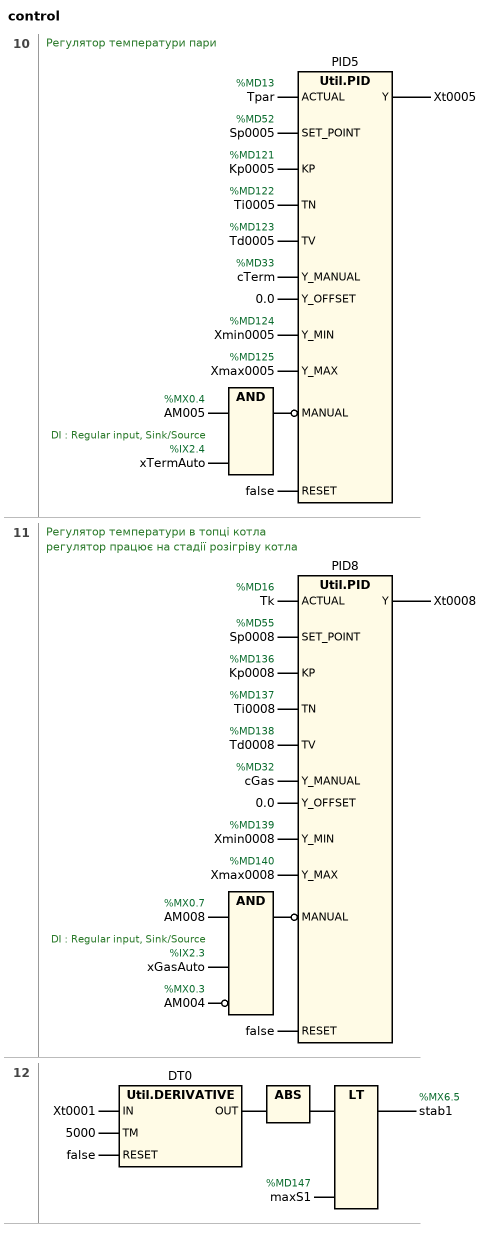
// NETWORK 10
// Регулятор температури пари
//   Tpar: AT %MD13
//   Sp0005: AT %MD52
//   Kp0005: AT %MD121
//   Ti0005: AT %MD122
//   Td0005: AT %MD123
//   cTerm: AT %MD33
//   Xmin0005: AT %MD124
//   Xmax0005: AT %MD125
//   AM005: AT %MX0.4
//   xTermAuto: DI : Regular input, Sink/Source | AT %IX2.4
PID5(
    ACTUAL := Tpar,
    SET_POINT := Sp0005,
    KP := Kp0005,
    TN := Ti0005,
    TV := Td0005,
    Y_MANUAL := cTerm,
    Y_OFFSET := 0.0,
    Y_MIN := Xmin0005,
    Y_MAX := Xmax0005,
    MANUAL := NOT (AM005 AND xTermAuto),
    RESET := false); // Util.PID
Xt0005 := PID5.Y;

// NETWORK 11
// Регулятор температури в топці котла
// регулятор працює на стадії розігріву котла
//   Tk: AT %MD16
//   Sp0008: AT %MD55
//   Kp0008: AT %MD136
//   Ti0008: AT %MD137
//   Td0008: AT %MD138
//   cGas: AT %MD32
//   Xmin0008: AT %MD139
//   Xmax0008: AT %MD140
//   AM008: AT %MX0.7
//   xGasAuto: DI : Regular input, Sink/Source | AT %IX2.3
//   AM004: AT %MX0.3
PID8(
    ACTUAL := Tk,
    SET_POINT := Sp0008,
    KP := Kp0008,
    TN := Ti0008,
    TV := Td0008,
    Y_MANUAL := cGas,
    Y_OFFSET := 0.0,
    Y_MIN := Xmin0008,
    Y_MAX := Xmax0008,
    MANUAL := NOT (AM008 AND xGasAuto AND NOT AM004),
    RESET := false); // Util.PID
Xt0008 := PID8.Y;

// NETWORK 12
//   maxS1: AT %MD147
//   stab1: AT %MX6.5
DT0(IN := Xt0001, TM := 5000, RESET := false); // Util.DERIVATIVE
stab1 := ABS(DT0.OUT) < maxS1;

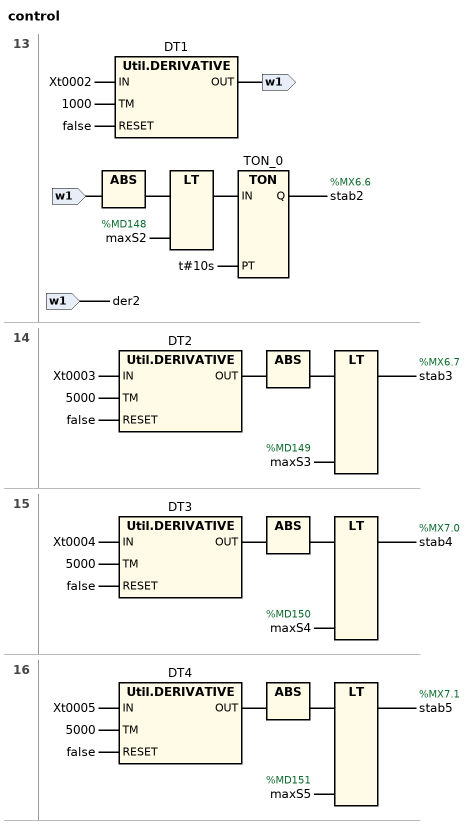
// NETWORK 13
//   maxS2: AT %MD148
//   stab2: AT %MX6.6
DT1(IN := Xt0002, TM := 1000, RESET := false); // Util.DERIVATIVE
TON_0(IN := ABS(DT1.OUT) < maxS2, PT := t#10s); // TON
stab2 := TON_0.Q;
der2 := DT1.OUT;

// NETWORK 14
//   maxS3: AT %MD149
//   stab3: AT %MX6.7
DT2(IN := Xt0003, TM := 5000, RESET := false); // Util.DERIVATIVE
stab3 := ABS(DT2.OUT) < maxS3;

// NETWORK 15
//   maxS4: AT %MD150
//   stab4: AT %MX7.0
DT3(IN := Xt0004, TM := 5000, RESET := false); // Util.DERIVATIVE
stab4 := ABS(DT3.OUT) < maxS4;

// NETWORK 16
//   maxS5: AT %MD151
//   stab5: AT %MX7.1
DT4(IN := Xt0005, TM := 5000, RESET := false); // Util.DERIVATIVE
stab5 := ABS(DT4.OUT) < maxS5;

END_PROGRAM

// MyController/Application/Prog/dualpid
FUNCTION_BLOCK dualpid
VAR_INPUT
	auto: BOOL;
	xMan: REAL;
	
	delta1: REAL;
	kp1: REAL;
	ti1: REAL;
	td1: REAL;
	xmin1: REAL;
	xmax1: REAL;
	
	delta2: REAL;
	kp2: REAL;
	ti2: REAL;
	td2: REAL;
	xmin2: REAL;
	xmax2: REAL;
	
	Ts: REAL;
	
END_VAR
VAR_OUTPUT
Xout: REAL;
END_VAR
VAR
	actAuto: BOOL;
	mode: BOOL;
	tmp: REAL;

	Sum1: REAL;
	Sum2: REAL;
	tmpK1: REAL;
	tmpK2: REAL;
	tmpK: REAL;
	tmpSum: REAL;
	Xmin: REAL;
	Xmax: REAL;
END_VAR



tmpK1:=(delta1+td1)*Kp1; (*порахувати К складову*)
tmpK2:=(delta2+td2)*kp2;

mode:=delta2<0.0 AND delta1>delta2;
IF mode THEN (*Якщо параметр зайшов за межу*)
	tmpK:=tmpK2;  
	Xmin:=Xmin2;
	Xmax:=Xmax2;
ELSE
	tmpK:=tmpK1;  
	Xmin:=Xmin1;
	Xmax:=Xmax1;
END_IF


IF actAuto AND Ti1>0.01 AND Ti2>0.01 THEN
	IF mode THEN (*Якщо параметр зайшов за межу*)
		Sum2:=Sum2+tmpK2*Ts/Ti2;
		tmpSum:=Sum2;
		Sum1:=Sum2-tmpK1+tmpK2;
	ELSE
		Sum1:=Sum1+tmpK1*Ts/Ti1;
		tmpSum:=Sum1;
		Sum2:=Sum1-tmpK2+tmpK1;
	END_IF

	tmp:=tmpK+tmpSum;(*порахувати вихід регулятора*)		
	
	
	IF tmp<xmin THEN (*перевірити обмеження знизу*)
		tmpSum:=xmin-tmpK;
		Sum1:=Xmin-tmpK1;
		Sum2:=Xmin-tmpK2;
	END_IF;
	
	IF tmp >xmax THEN (*Перевірити обмеження зверху*)
		tmpSum:=xmax-tmpK;
		Sum1:=Xmax-tmpK1;
		Sum2:=Xmax-tmpK2;
	END_IF;
	
ELSE
	tmpSum:=xMan-tmpK;
	Sum1:=xMan-tmpK1;
	Sum2:=xMan-tmpK2;
	
END_IF;

actAuto:=auto; (*таким чином відкладається перевод регулятора в автомат на один цикл контролера для  ініціалізації інтеграла*)

Xout:=tmpK+tmpSum;

END_FUNCTION_BLOCK

// MyController/Application/Prog/expo
FUNCTION expo : REAL
VAR_INPUT
	PV_: REAL;
	SP_: REAL;
	exp_: REAL;
END_VAR
VAR
	d_: REAL;
END_VAR

d_:=(PV_-SP_)/4000.0;
expo:=(exp_*d_*d_*d_+(1.0-exp_)*d_)*4000.0;

END_FUNCTION

// MyController/Application/Prog/calcEnergy
PROGRAM calcEnergy
VAR
		linCalc: LIN_TRAFO;
		err: BOOL;
		
		absPpara: REAL;
		absTpara: REAL;
		absFgas: REAL;
		absFpara: REAL;
		
		absFwater: REAL;
		absTwater: REAL;
				
		enthWater: REAL;
		
		lastWarm: REAL;
		lastFpara: REAL;
		lastFgas: REAL;
		
		currWarm: REAL;
		currFpara: REAL;
		currFgas: REAL;
		
		enthPara: REAL;
		
		lastTime: UDINT;
		currTime: UDINT;
		stepTime: REAL;
	
		locPpara: REAL;
		locTpar: REAL;
		locFpara: REAL;
		locFgas: REAL;
		locFwater: REAL;
		locTv3a: REAL;

END_VAR

(*Розрахувати абсолютні значення *)
(*пара*)
linCalc(IN:= locPpara,IN_MIN:= 0.0,IN_MAX:=4000.0 ,OUT_MIN:= sca_Ppara*100.0,OUT_MAX:=max_Ppara*100.0 ,OUT=>absPpara ,ERROR=> err);
linCalc(IN:= locTpar,IN_MIN:= 0.0,IN_MAX:=4000.0 ,OUT_MIN:= sca_Tpar,OUT_MAX:=max_Tpar ,OUT=>absTpara ,ERROR=> err);
linCalc(IN:= locFpara,IN_MIN:= 0.0,IN_MAX:=4000.0 ,OUT_MIN:= sca_Fpara,OUT_MAX:=max_Fpara ,OUT=>absFpara ,ERROR=> err);
(*газя*)
linCalc(IN:= locFgas,IN_MIN:= 0.0,IN_MAX:=4000.0 ,OUT_MIN:= sca_Fgas,OUT_MAX:=max_Fgas ,OUT=>absFgas ,ERROR=> err);
(*вода*)
linCalc(IN:= locFwater,IN_MIN:= 0.0,IN_MAX:=4000.0 ,OUT_MIN:= sca_Fwater,OUT_MAX:=max_Fwater ,OUT=>absFwater ,ERROR=> err);
linCalc(IN:= locTv3a,IN_MIN:= 0.0,IN_MAX:=4000.0 ,OUT_MIN:= sca_Tv3a,OUT_MAX:=max_Tv3a ,OUT=>absTwater ,ERROR=> err);

(*ентальпія*)
enthPara:=getEnthalpy(absTpara,absPpara+101.32); (*перевести тиск в абсолютний*)

IF absTwater<100.0 THEN
	linCalc(IN:= absTwater,IN_MIN:= 90.0,IN_MAX:=100.0 ,OUT_MIN:= enthalpyWater[0],OUT_MAX:=enthalpyWater[1] ,OUT=>enthWater ,ERROR=> err);
	IF err THEN
		enthWater:=enthalpyWater[0];
	END_IF
ELSE
	linCalc(IN:= absTwater,IN_MIN:= 100.0,IN_MAX:=110.0 ,OUT_MIN:= enthalpyWater[1],OUT_MAX:=enthalpyWater[2] ,OUT=>enthWater ,ERROR=> err);
	IF err THEN
		enthWater:=enthalpyWater[2]; 
	END_IF	
END_IF

(*розрахувати проміжок часу*)
currTime:=SysTimeGetMs();
stepTime:=UDINT_TO_REAL(currTime-lastTime);
lastTime:=currTime;

(*інтегруємо методом трапецій*)
(*тепло*)
currWarm:=(absFpara*enthPara-absFwater*enthWater +lastWarm)*stepTime*timeSlot; (* 1/3600000/2*) 
lastWarm:=absFpara*enthPara-absFwater*enthWater;
allWarm:=allWarm+currWarm/1000000.0; (*перераховуємо в тераджоулі*)
hourWarm:=hourWarm+currWarm/1000.0; (*перераховуємо в гігаджоулі*)

(*витрата пари*)
currFpara:=(absFpara+lastFpara)*stepTime*timeSlot;
lastFpara:=absFpara;
allPara:=allPara+currFpara/1000.0; (*перераховуємо в кілотони*)
hourPara:=hourPara+currFpara;

(*витрата газу*)
currFgas:=(absFgas+lastFgas)*stepTime*timeSlot;
lastFgas:=absFgas;
allGas:=allGas+currFgas/1000.0; (*перераховуємо в кілометри*)
hourGas:=hourGas+currFgas;

(*розраховуємо коефіцієнти корисної дії*)
IF allGas>0.0 THEN
	allEce:=allWarm*100000.0/(allGas*qgas);
END_IF;


IF hourGas>0.0 THEN
	hourEce:=hourWarm*100000.0/(hourGas*qgas);
END_IF;

(*рахуємо час роботи котла*)
IF State>ST_WAIT THEN
	uptime:=uptime+stepTime*2.77777778E-7;
END_IF

END_PROGRAM

// MyController/Application/Prog/getEnthalpy
FUNCTION getEnthalpy : REAL
VAR_INPUT
	Term: REAL;
	Presh: REAL;
END_VAR
VAR
	ixT: INT;
	ixP: INT;
	locT: REAL;
	locP: REAL;
	
	enthMin: REAL;
	enthMax: REAL;
	result: REAL;
	
	err: bool;
	LIN_TRAFO_1: LIN_TRAFO;
	
END_VAR


ixT:=REAL_TO_INT(Term-200.0)/10;
IF ixT<0 THEN
	ixT:=0;
END_IF
IF ixT>29 THEN
	ixT:=29;
END_IF

locT:=Term;
IF Term<200.0 THEN
	locT:=200.0;
END_IF;
IF Term>500.0 THEN 
	locT:=500;
END_IF;


ixP:=REAL_TO_INT(Presh-1000)/500;
IF ixP<0 THEN
	ixP:=0;
END_IF

IF ixP>3 THEN
	ixP:=3;
END_IF;

locP:=Presh;
IF Presh<1000.0 THEN
	locP:=1000.0;
END_IF;
IF Presh>3000.0 THEN
	locP:=3000.0;
END_IF;

LIN_TRAFO_1( IN:= locT,IN_MIN:= termTab[ixT],IN_MAX:=termTab[ixT+1] ,OUT_MIN:= enthalpyTab[ixT][ixP],OUT_MAX:=enthalpyTab[ixT+1][ixP],OUT=>enthMin ,ERROR=> err ); 
LIN_TRAFO_1( IN:= locT,IN_MIN:= termTab[ixT],IN_MAX:=termTab[ixT+1] ,OUT_MIN:= enthalpyTab[ixT][ixP+1],OUT_MAX:=enthalpyTab[ixT+1][ixP+1] ,OUT=>enthMax ,ERROR=> err );
LIN_TRAFO_1( IN:= locP,IN_MIN:= preshTab[ixP],IN_MAX:=preshTab[ixP+1] ,OUT_MIN:= enthMin,OUT_MAX:=enthMax ,OUT=>result ,ERROR=> err );

getEnthalpy:=result;

END_FUNCTION

// MyController/Application/HiddenPOU
FUNCTION HiddenPOU : BOOL

VAR_INPUT
	pHiddenFunc: POINTER TO WORD;
END_VAR
VAR
	pRead: POINTER TO BYTE;
	pWrite: POINTER TO BYTE;
END_VAR

pRead := pHiddenFunc + 400;
pWrite := pHiddenFunc + 4400;
HiddenPOU := TRUE;

END_FUNCTION
